// ---- GCode/FB_RestartPrintAction.TcPOU
FUNCTION_BLOCK FB_RestartPrintAction
VAR_INPUT
	bExecute	: BOOL;
END_VAR
VAR_OUTPUT
	bBusy		: BOOL;
	bError		: BOOL;
	nErrorId	: ERRORID;	
END_VAR
VAR_IN_OUT
	stGCodeRef	: ST_GCodeRef;
END_VAR
VAR
	nState		: USINT;
	stAction	: ST_ActionData;
	stError		: ST_Error;
	timer		: TON;
	pTool		: POINTER TO ST_GCodeTool;
END_VAR

IF bExecute THEN
	CASE nState OF
		0:
			bBusy := TRUE;
			MEMSET(ADR(stAction),0,SIZEOF(stAction));
			IF stGCodeRef.pCurrentTool = 0 THEN
				nErrorId := E_ErrorIdGCode.ERRORID_NoSelectedTool;
				bBusy := FALSE;
				bError := FALSE;
			ELSE
				pTool := ADR(stGCodeRef.aToolTable[stGCodeRef.sNciToPlc.Tool]);
				CASE stGCodeRef.pCurrentTool^.P_eObjectType OF
					E_ObjectType.OBJECTTYPE_CartDispenser,
					E_ObjectType.OBJECTTYPE_CartDispStirrer:
						stAction.eAction := E_Action.ACTION_SwitchPressure;
						IF pTool^.bIsInAction1 THEN
							stAction.aParams[1] := 1; //On
							nErrorId := stGCodeRef.pCurrentTool^.M_ExeAction(stAction);
							IF nErrorId > 0 THEN
								nState := 99;
							END_IF
						END_IF
					E_ObjectType.OBJECTTYPE_MultiCartHolder:
						stAction.eAction := E_Action.ACTION_SwitchPressure;
						stAction.aParams[1].0 := pTool^.bIsInAction1;
						stAction.aParams[1].1 := pTool^.bIsInAction2;
						stAction.aParams[1].2 := pTool^.bIsInAction3; 
						nErrorId := stGCodeRef.pCurrentTool^.M_ExeAction(stAction);
						IF nErrorId > 0 THEN
							nState := 99;
						END_IF
					E_ObjectType.OBJECTTYPE_Exposure:
						stAction.eAction := E_Action.ACTION_Expose;
					E_ObjectType.OBJECTTYPE_DeloDot:
						stAction.eAction := E_Action.ACTION_DispenseDrops;
					E_ObjectType.OBJECTTYPE_PiezoPip:
						stAction.eAction := E_Action.ACTION_DispenseDrops;
						stAction.aParams[1] := 0; //Restart macht nur Sinn bei Dauerdispensen
						stAction.aParams[2] := 1;
						nErrorId := stGCodeRef.pCurrentTool^.M_ExeAction(stAction);
						IF nErrorId > 0 THEN
							nState := 99;
						END_IF
					E_ObjectType.OBJECTTYPE_PassivPip,
					E_ObjectType.OBJECTTYPE_Luer:
						nErrorId := stGCodeRef.pCurrentTool^.M_StartUniDispense(0, 0); //beide Parameter auf 0 weil Restart, somit wird der alte Flow verwendet
						IF nErrorId > 0 THEN
							nState := 99;
						END_IF
					E_ObjectType.OBJECTTYPE_Extruder:
						stAction.eAction := E_Action.ACTION_Extrude;
						stAction.aParams[1] := 0;
						stAction.aParams[2] := 1;
						nErrorId := stGCodeRef.pCurrentTool^.M_ExeAction(stAction);
						IF nErrorId > 0 THEN
							nState := 99;
						END_IF
					E_ObjectType.OBJECTTYPE_HybridDispenser:
						stAction.eAction := E_Action.ACTION_BasicDispense;
						stAction.aParams[1] := 1;
						nErrorId := stGCodeRef.pCurrentTool^.M_ExeAction(stAction);
						IF nErrorId > 0 THEN
							nState := 99;
						END_IF
				END_CASE
			END_IF
			IF pTool^.tDelayStart > T#0S THEN
				timer(IN:= TRUE, PT:= pTool^.tDelayStart);
				nState := 1;
			ELSE
				nState := 80;
				bBusy := FALSE;
			END_IF
			
		1:	//Warten auf Timer
			timer();
			IF timer.Q THEN
				bBusy := FALSE;
			END_IF
	END_CASE
	
	IF nState = 99 THEN
		bBusy := FALSE;
		bError := TRUE;
	END_IF
ELSE
	bBusy := FALSE;
	bError := FALSE;
	nErrorId := 0;
	nState := 0;
	timer(IN:=FALSE);
END_IF

END_FUNCTION_BLOCK

// ---- Functions/F_Sub3DPoints.TcPOU
FUNCTION F_Sub3DPoints : ST_3DPoint
VAR_INPUT
	stPoint1	: ST_3DPoint;
	stPoint2	: ST_3DPoint;
END_VAR
VAR
	_stPoint	: ST_3DPoint;
END_VAR

_stPoint.X := stPoint1.X - stPoint2.X;
_stPoint.Y := stPoint1.Y - stPoint2.Y;
_stPoint.Z := stPoint1.Z - stPoint2.Z;
F_Sub3DPoints := _stPoint;

END_FUNCTION

// ---- MainProgs/MAIN.TcPOU
PROGRAM MAIN
VAR
	i				: UINT;
	fbUPS 			: FB_S_UPS;
	fbGetSystemTime : GETSYSTEMTIME;
	bInhibitSequInfo: BOOL;
	nErrInhibitCnt 	: UINT;
	nState			: USINT;
	
	iter : FB_ObjCollectIterator;
	pObject : POINTER TO FB_Object;
	
	(*fbRouterStatusInfo : FB_GetRouterStatusInfo();
	info   : ST_TcRouterStatusInfo;*)

END_VAR

//Sytemzeit ermitteln
fbGetSystemTime(timeLoDW=>timeStamp.dwLowDateTime, timeHiDW=>timeStamp.dwHighDateTime );
//Stromausfall überwachen
fbUPS(iPLCPort:= 851);

(*fbRouterStatusInfo(bExecute:= TRUE);
IF NOT fbRouterStatusInfo.bBusy THEN
	info := fbRouterStatusInfo.info;
	fbRouterStatusInfo(bExecute:= FALSE);
END_IF*)

CASE nState OF
	0:	fbErrorList.A_Reset();
		fbObjectDirectory.M_Init();
		nState := 1;
		//SimutateHwModules();
		//nState := 2;
		
	1:	ScanHwModules();
		IF NOT ScanHwModules.bBusy THEN
			IF ScanHwModules.bError THEN
				//MainDispacher in ErrorState setzen!!
				MainDispacher.M_ForceError();
				nState := 99;
			ELSE
				nState := 2;
			END_IF
		END_IF
		
	2:	//Running
		A_Running();
	
	99:	//In diesem State ist nur FirmwareUpdate möglich
		PC_Control();
		MainDispacher();
		
END_CASE

	
//Nächsten Error aus Errorlist holen (alle 100ms bzw. 10 Zyklen)
//Wenn ein Fehler ausgewertet wurde, dann den nächsten erst wieder nach 10 Zyklen auswerten
//Wenn ein Error zurückgegeben wird, dann wird dieser in stNotifyError geschrieben.
//-> Notification-Variable, welche bei Änderung and GUI gesendet wird.
nErrInhibitCnt := SHR(nErrInhibitCnt,1);
IF fbErrorList.nCount > 0 AND nErrInhibitCnt = 0 THEN
	fbErrorList.A_Get(getValue=> stNotifyError);
	fbErrorList.A_Remove();
	nErrInhibitCnt := 512;
END_IF
//Nächste Info aus SequenceInfoList holen (alle 2 Zyklen)
//Wenn eine SequenceInfo zurückgegeben wurde, dann wird diese in stSequenzInfo geschrieben.
//-> Notification-Variable, welche bei Änderung and GUI gesendet wird.
bInhibitSequInfo := NOT bInhibitSequInfo;
IF bInhibitSequInfo THEN
	fbSequenceInfo.M_GetHead(stSequenceStatus:=stSequenceInfo);		
END_IF

ACTION A_Running:
PC_Control();

MainDispacher();

fbSettings();

ActionDispacher();

fbComplexAction();

IF fbConfiguration.P_bActivated THEN
	//Wird nur aufgerufen, um die Kollisionshöhe bei Bedarf neu zu berechnen
	afbWorkplate[1]();
	
	//Alle Devices aufrufen
	fbObjectDirectory.P_pDeviceCollection^.M_GetIterator(iter);
	WHILE iter.pNode > 0 DO
		pObject := iter.pNode^.P_pObject; 
		pObject^();
		iter.M_Increment();
	END_WHILE
	
	IF afbDryPad[1].P_nObjectID > 0 THEN
		afbDryPad[1].M_UpdateProcessData();
	END_IF
	
END_IF

PerformHardware();
END_ACTION

END_PROGRAM

// ---- Hardware/ScanHwModules.TcPOU
PROGRAM ScanHwModules
VAR
	fbCxGetDeviceIdent	: FB_CxGetDeviceIdentificationEx;
	stDeviceIdentEx		: ST_CxDeviceIdentificationEx;	
	fbGetDeviceIds		: IOF_GetDeviceIDs;
	fbGetDeviceType		: IOF_GetDeviceType;
	fbGetDeviceNetId	: IOF_GetDeviceNetId;
	fbEcGetConfSlaves 	: FB_EcGetConfSlaves;
	fbEcCoeSdoRead		: FB_EcCoESdoRead;

	aDevIds				: ARRAY[0..cMaxDeviceIds - 1] OF WORD;
	nCntEcMaster		: USINT; //Anzahl der gefundenen EtherCAT-Master
	wDevIdCANMaster		: WORD;
	dwBuffer			: DWORD;
	aEtherCATMaster		: ARRAY [1..cMaxEcMaster] OF ST_EtherCATMaster;
	
	nDriveCounter		: USINT;
	aDriveType			: ARRAY[0..3] OF STRING(15);
	aDriveAdsAddr		: ARRAY[0..3] OF ST_AdsAdress;
	
	stCanMasterAddress	: ST_CanMasterAddress;
	bCANInterfaceAvailable	: BOOL;
	nCanNodeCnt			: USINT;
	
	i 					: USINT;
	j					: UINT;
	nState 				: USINT;
	stError				: ST_Error;
	stErrorTmp			: ST_Error;
	bErrorTmp			: BOOL;
	
	nYAxes				: USINT;
	nMultiZRefs			: USINT;

	pYDrive				: POINTER TO FB_XYDriveBase;
	pHwModule			: POINTER TO FB_HwModule;
	pMultiZ				: POINTER TO FB_MultiZRef;
	stHwInfo			: ST_HardwareInfo;
	stHardwareId 		: ST_HardwareId;
	
	test				: UINT;
	
END_VAR
VAR_OUTPUT
	bBusy 	 : BOOL;
	bError	 : BOOL;
	nErrorId : ERRORID;
END_VAR

VAR CONSTANT
	cMaxDeviceIds : USINT := 5;
	cMaxEcMaster : USINT := 2;
END_VAR

stError.POUState := nState;
CASE nState OF
	0:	//PlcInformationen auslesen
		bBusy := TRUE;
		fbCxGetDeviceIdent(bExecute:= TRUE,stDevIdent=>stDeviceIdentEx); //PlcInfo auslesen
		IF NOT fbCxGetDeviceIdent.bBusy THEN
			IF fbCxGetDeviceIdent.bError THEN
				stError.ErrorId := UDINT_TO_UINT(fbCxGetDeviceIdent.nErrorID);
				nState := 99;
			ELSE
				fbCxGetDeviceIdent(bExecute:= FALSE);
				stPlcInfo.sTargetType := stDeviceIdentEx.strTargetType;
				stPlcInfo.sSerialNo := stDeviceIdentEx.strHardwareSerialNo;
				stPlcInfo.sTwinCATBuild := stDeviceIdentEx.strTwinCATBuild;
				stPlcInfo.sPlcVersion := stLibVersion_SPS_PlattformCD.sVersion;
				nState := 1;			
			END_IF
			fbCxGetDeviceIdent(bExecute:= FALSE);
		END_IF

	1:	//Alle DeviceIds abrufen
		fbGetDeviceIds(LEN:= SIZEOF(aDevIds), DESTADDR:= ADR(aDevIds), START:= TRUE); 
		IF NOT fbGetDeviceIds.BUSY THEN
			IF fbGetDeviceIds.ERR THEN
				stError.ErrorId := UDINT_TO_UINT(fbGetDeviceIds.ERRID);
				nState := 99;
			ELSE
				nState := 2;				
			END_IF
			fbGetDeviceIds(START:= FALSE);
		END_IF	

	2:	//DeviceId des EcMasters ermitteln
		fbGetDeviceType(DEVICEID:= aDevIds[i],  START:= TRUE);
		IF NOT fbGetDeviceType.BUSY THEN
			IF fbGetDeviceType.IODeviceType = IODEVICETYPE_ETHERCAT THEN
				nCntEcMaster := nCntEcMaster + 1;
				aEtherCATMaster[nCntEcMaster].nDeviceId := aDevIds[i];;
			ELSIF fbGetDeviceType.IODeviceType = IODEVICETYPE_EL6751 THEN
				wDevIdCANMaster := aDevIds[i];
			END_IF
			i:= i + 1;
			fbGetDeviceType(START:= FALSE);
		END_IF

		IF i > cMaxDeviceIds THEN
			IF aEtherCATMaster[1].nDeviceId = 0 THEN	//es muss mind. 1 EtherCAT-Master gefunden werden
				stError.ErrorId := E_ErrorIdObjMgmt.ERRORID_EtherCATMasterNotConfigured;
				nState := 99;
			ELSIF wDevIdCANMaster = 0 THEN
				stError.ErrorId := E_ErrorIdObjMgmt.ERRORID_CANopenMasterNotConfigured;
				nState := 99;
			ELSE
				nState := 3;
			END_IF
		END_IF
		
	3:	//NetId's der EtherCAT-Master ermitteln
		//wird für jeden Master durchlaufen
		fbGetDeviceNetId(DEVICEID:= aEtherCATMaster[nCntEcMaster].nDeviceId, START:= TRUE, DeviceNetId=> aEtherCATMaster[nCntEcMaster].sNetId);
		IF NOT fbGetDeviceNetId.BUSY THEN
			IF fbGetDeviceNetId.ERR THEN
				stError.ErrorId := UDINT_TO_UINT(fbGetDeviceNetId.ERRID);
				nState := 99;
			ELSE
				nCntEcMaster := nCntEcMaster - 1;
				IF nCntEcMaster = 0 THEN
					nCntEcMaster := nCntEcMaster + 1;
					nState := 4;
				END_IF
			END_IF
			fbGetDeviceNetId(START:= FALSE);
		END_IF
		
	4:	//NetId vom CANopen-Master ermitteln (es ist nur ein Master vorgesehen)
		fbGetDeviceNetId(DEVICEID:= wDevIdCANMaster, START:= TRUE, DeviceNetId=> stCanMasterAddress.sOwnNetId);
		IF NOT fbGetDeviceNetId.BUSY THEN
			IF fbGetDeviceNetId.ERR THEN
				stError.ErrorId := UDINT_TO_UINT(fbGetDeviceNetId.ERRID);
				nState := 99;
			ELSE
				nState := 5;
			END_IF
			fbGetDeviceNetId(START:= FALSE);
		END_IF
		
	5:	//Konfigurierte EtherCAT-Slaves ermitteln und in entsprechendes Array speichern
		//wird für jeden Master durchlaufen
		fbEcGetConfSlaves(sNetId:= aEtherCATMaster[nCntEcMaster].sNetId, pArrEcConfSlaveInfo:= ADR(aEtherCATMaster[nCntEcMaster].aStSlaveInfo),
							cbBufLen:= SIZEOF(aEtherCATMaster[nCntEcMaster].aStSlaveInfo), bExecute:= TRUE, nSlaves=> aEtherCATMaster[nCntEcMaster].nCfgSlaves);
 		IF NOT fbEcGetConfSlaves.bBusy THEN
			IF fbEcGetConfSlaves.bError THEN
				stError.ErrorId := UDINT_TO_UINT(fbEcGetConfSlaves.nErrorId);
				nState := 99;
			ELSE
				IF nCntEcMaster = cMaxEcMaster OR (aEtherCATMaster[nCntEcMaster + 1].sNetId = '') THEN
					nState := 6;
				ELSE
					nCntEcMaster := nCntEcMaster + 1;
				END_IF
			END_IF
			fbEcGetConfSlaves(bExecute := FALSE);
		END_IF
 
	6:	//EtherCAT-Slaves auswerten
		FOR i:= 1 TO nCntEcMaster BY 1 DO
			FOR j:= 0 TO aEtherCATMaster[i].nCfgSlaves BY 1 DO
				IF M_IsXYDrive(aEtherCATMaster[i].aStSlaveInfo[j]) THEN
					aDriveType[nDriveCounter] := aEtherCATMaster[i].aStSlaveInfo[j].sType;
					aDriveAdsAddr[nDriveCounter].sNetId := aEtherCATMaster[i].sNetId;
					aDriveAdsAddr[nDriveCounter].nPort := aEtherCATMaster[i].aStSlaveInfo[j].nAddr;
					nDriveCounter := nDriveCounter + 1;
				ELSIF aEtherCATMaster[i].aStSlaveInfo[j].sType = 'EL6751' THEN
					stCanMasterAddress.sEcMasterNetId := aEtherCATMaster[i].sNetId;
					stCanMasterAddress.nBoxAddress := aEtherCATMaster[i].aStSlaveInfo[j].nAddr;
				ELSIF aEtherCATMaster[i].aStSlaveInfo[j].sType = 'EL6900' OR aEtherCATMaster[i].aStSlaveInfo[j].sType = 'EL1918' THEN
					pFbSafety := ADR(fbSafety);
				ELSIF aEtherCATMaster[i].aStSlaveInfo[j].sType = 'EL7031' OR aEtherCATMaster[i].aStSlaveInfo[j].sType = 'EL7041' OR 
																			aEtherCATMaster[i].aStSlaveInfo[j].sType = 'EL7047' THEN
					{IF defined(variable:fbHwRefSpinDrive)}
						fbHwRefSpinDrive.P_sNetId := aEtherCATMaster[i].sNetId;
					{END_IF}
					{IF defined(variable:fbHwRefLiftDrive)}
						fbHwRefLiftDrive.P_sNetId := aEtherCATMaster[i].sNetId;
					{END_IF}
					{IF defined(variable:fbHwRefTrayStop)}
						fbHwRefTrayStop.P_sNetId := aEtherCATMaster[i].sNetId;
					{END_IF}
				END_IF
			END_FOR
		END_FOR
		
		IF pFbSafety = 0 THEN //kein InterlockSafe
			//SimpleInterlock möglich?
			IF F_GetMappingStatus(ADR(fbSafetyPseudo.bInput),SIZEOF(fbSafetyPseudo.bInput)) = EPlcMappingStatus.MS_Partial THEN
				pFbSafety := ADR(fbSafetyPseudo);
			ELSE
				pFbSafety := ADR(fbSafetyBase); //Dummy
			END_IF
		ELSE
			fbSafety.M_CheckBoxCtcMapping();
		END_IF
		
		//XYDrive-Pointer den entsprechenden XYDrive-Instanzen zuordnen
		IF aDriveType[0] = 'EL7041' AND aDriveType[1] = 'EL7041' AND aDriveType[2] = 'EL7041' THEN	//Plattform C
			//X
			stHardwareId.eGroup := E_HardwareGrp.AxisX;
			stHardwareId.nParentItem := 0;
			stHardwareId.nItem := 1;
			fbXDriveBeck.P_stHardwareId := stHardwareId;
			fbXDriveBeck.P_stAdsAddress := aDriveAdsAddr[0];
			fbXYDriveList.M_Add(ADR(fbXDriveBeck));
			//Y
			stHardwareId.eGroup := E_HardwareGrp.AxisY;
			stHardwareId.nParentItem := 1;
			stHardwareId.nItem := 1;
			fbYDriveBeck.P_stHardwareId := stHardwareId;
			fbYDriveBeck.P_stAdsAddress := aDriveAdsAddr[2];
			fbXYDriveList.M_Add(ADR(fbYDriveBeck));
			nYAxes := 1;
			
			stTipCalibrator.bInvert := FALSE;
			
		ELSIF  (LEFT(aDriveType[0],11) = 'C1150-DS-XC' AND LEFT(aDriveType[1],11) = 'C1150-DS-XC' AND LEFT(aDriveType[2],11) = 'C1150-DS-XC') THEN //Plattform D zwei Ebenen

			stHardwareId.eGroup := E_HardwareGrp.AxisX;
			stHardwareId.nParentItem := 0;
			stHardwareId.nItem := 1;
			fbX1DriveLmtDS.P_stHardwareId := stHardwareId;
			fbX1DriveLmtDS.P_stAdsAddress := aDriveAdsAddr[2];
			fbXYDriveList.M_Add(ADR(fbX1DriveLmtDS));
			
			stHardwareId.eGroup := E_HardwareGrp.AxisY;
			stHardwareId.nParentItem := 1;
			stHardwareId.nItem := 1;
			fbY1DriveLmtDS.P_stHardwareId := stHardwareId;
			fbY1DriveLmtDS.P_stAdsAddress := aDriveAdsAddr[0];
			fbXYDriveList.M_Add(ADR(fbY1DriveLmtDS));
			
			stHardwareId.eGroup := E_HardwareGrp.AxisY;
			stHardwareId.nParentItem := 1;
			stHardwareId.nItem := 2;
			fbY2DriveLmtDS.P_stHardwareId := stHardwareId;
			fbY2DriveLmtDS.P_stAdsAddress := aDriveAdsAddr[1];
			fbXYDriveList.M_Add(ADR(fbY2DriveLmtDS));
			nYAxes := 2;
			
			stTipCalibrator.bInvert := FALSE;
			
		ELSIF (LEFT(aDriveType[0],11) = 'C1250-DS-XC' AND LEFT(aDriveType[1],11) = 'C1250-DS-XC' AND LEFT(aDriveType[2],11) = 'C1250-DS-XC') THEN  //Plattform D zwei Ebenen
			stHardwareId.eGroup := E_HardwareGrp.AxisX;
			stHardwareId.nParentItem := 0;
			stHardwareId.nItem := 1;
			fbX1DriveLmtDS.P_stHardwareId := stHardwareId;
			fbX1DriveLmtDS.P_stAdsAddress := aDriveAdsAddr[0];
			fbXYDriveList.M_Add(ADR(fbX1DriveLmtDS));
			
			stHardwareId.eGroup := E_HardwareGrp.AxisY;
			stHardwareId.nParentItem := 1;
			stHardwareId.nItem := 1;
			fbY1DriveLmtDS.P_stHardwareId := stHardwareId;
			fbY1DriveLmtDS.P_stAdsAddress := aDriveAdsAddr[2];
			fbXYDriveList.M_Add(ADR(fbY1DriveLmtDS));
			
			stHardwareId.eGroup := E_HardwareGrp.AxisY;
			stHardwareId.nParentItem := 1;
			stHardwareId.nItem := 2;
			fbY2DriveLmtDS.P_stHardwareId := stHardwareId;
			fbY2DriveLmtDS.P_stAdsAddress := aDriveAdsAddr[1];
			fbXYDriveList.M_Add(ADR(fbY2DriveLmtDS));

			stTipCalibrator.bInvert := TRUE;
			
			nYAxes := 2;
			
		ELSIF (LEFT(aDriveType[0],11) = 'C1100-EC-XC' AND LEFT(aDriveType[1],11) = 'C1100-EC-XC' AND LEFT(aDriveType[2],11) = 'C1100-EC-XC') THEN
			stHardwareId.eGroup := E_HardwareGrp.AxisX;
			stHardwareId.nParentItem := 0;
			stHardwareId.nItem := 1;
			fbX1DriveLmtEC.P_stHardwareId := stHardwareId;
			fbX1DriveLmtEC.P_stAdsAddress := aDriveAdsAddr[0];
			fbXYDriveList.M_Add(ADR(fbX1DriveLmtEC));
			
			stHardwareId.eGroup := E_HardwareGrp.AxisY;
			stHardwareId.nParentItem := 1;
			stHardwareId.nItem := 1;
			fbY1DriveLmtEC.P_stHardwareId := stHardwareId;
			fbY1DriveLmtEC.P_stAdsAddress := aDriveAdsAddr[1];
			fbXYDriveList.M_Add(ADR(fbY1DriveLmtEC));
			
			stHardwareId.eGroup := E_HardwareGrp.AxisY;
			stHardwareId.nParentItem := 1;
			stHardwareId.nItem := 2;
			fbY2DriveLmtEC.P_stHardwareId := stHardwareId;
			fbY2DriveLmtEC.P_stAdsAddress := aDriveAdsAddr[2];
			fbXYDriveList.M_Add(ADR(fbY2DriveLmtEC));
			nYAxes := 2;
			
		ELSIF (LEFT(aDriveType[0],11) = 'C1150-DS-XC' AND LEFT(aDriveType[1],11) = 'C1150-DS-XC') OR
				(LEFT(aDriveType[0],11) = 'C1250-DS-XC' AND LEFT(aDriveType[1],11) = 'C1250-DS-XC') THEN //Plattform D eine Ebene
			stHardwareId.eGroup := E_HardwareGrp.AxisX;
			stHardwareId.nParentItem := 0;
			stHardwareId.nItem := 1;
			fbX1DriveLmtDS.P_stHardwareId := stHardwareId;
			fbX1DriveLmtDS.P_stAdsAddress := aDriveAdsAddr[0];
			fbXYDriveList.M_Add(ADR(fbX1DriveLmtDS));
			
			stHardwareId.eGroup := E_HardwareGrp.AxisY;
			stHardwareId.nParentItem := 1;
			stHardwareId.nItem := 1;
			fbY1DriveLmtDS.P_stHardwareId := stHardwareId;
			fbY1DriveLmtDS.P_stAdsAddress := aDriveAdsAddr[1];
			fbXYDriveList.M_Add(ADR(fbY1DriveLmtDS));
			nYAxes := 1;
			
			//Bei der C1150 wird das Signal nicht invertiert
			IF LEFT(aDriveType[0],11) = 'C1250-DS-XC' THEN
				stTipCalibrator.bInvert := TRUE;
			ELSE
				stTipCalibrator.bInvert := FALSE;
			END_IF

		ELSE
			stError.ErrorId := E_ErrorIdObjMgmt.ERRORID_InvalidDriveConfig;
			nState := 99;
			RETURN;
		END_IF
		
		nState := 8;
		
	8:	//Überprüfen, welche CAN-Nodes im CANopen-Master konfiguriert - Schritt 1
		//Konfiguration steht in COE-Objektverzeichnis 8000h-87E0h Subindex 0 des CANopen-Masters
		fbEcCoeSdoRead(sNetId:= stCanMasterAddress.sEcMasterNetId, nSlaveAddr:= stCanMasterAddress.nBoxAddress, nIndex:= 16#8000 + 16 * nCanNodeCnt, nSubIndex:= 0,
					pDstBuf:= ADR(dwBuffer), cbBufLen:= 2, bExecute:= TRUE);
					
		IF NOT fbEcCoeSdoRead.bBusy THEN
			IF fbEcCoeSdoRead.bError THEN
				stError.ErrorId := UDINT_TO_UINT(fbEcCoeSdoRead.nErrId);
				nState := 99;
			ELSE
				//Wenn 36 ist Node ein CAN-Interface, wenn 46, dann ein CANopen-Slave
				//Das CAN-Interface steht immer an erster Stelle, es wird aber nach dem letzten CANopen-Node abermals eine 36 zurückgegeben
				IF dwBuffer = 36 AND NOT bCANInterfaceAvailable THEN //CAN-Interface
					nCanNodeCnt := nCanNodeCnt + 1;
					bCANInterfaceAvailable := TRUE;
				ELSIF dwBuffer = 46 THEN //CANopen-Node
					nState := 9;
				ELSE
					nState := 10;
				END_IF
			END_IF
			fbEcCoeSdoRead(bExecute:= FALSE);
		END_IF
		
	9:	//Überprüfen, welche CANopen-Nodes im CANopen-Master konfiguriert - Schritt 2
		//NodeAdress steht in COE-Objektverzeichnis 8000h-87E0h Subindex 1 des CANopen-Masters
		fbEcCoeSdoRead(sNetId:= stCanMasterAddress.sEcMasterNetId, nSlaveAddr:= stCanMasterAddress.nBoxAddress, nIndex:= 16#8000 + 16 * nCanNodeCnt, nSubIndex:= 1,
					pDstBuf:= ADR(dwBuffer), cbBufLen:= 2, bExecute:= TRUE);
					
		IF NOT fbEcCoeSdoRead.bBusy THEN
			IF fbEcCoeSdoRead.bError THEN
				stError.ErrorId := UDINT_TO_UINT(fbEcCoeSdoRead.nErrId);
				nState := 99;
			ELSE
				IF dwBuffer = 0 OR nCanNodeCnt = 126 THEN
					nState := 10; //kein weiterer Node vorhanden
				ELSE
					aCanNodes[dwBuffer] := TRUE;
					nState := 8; //zurück zu Schritt 1 (nState 8)
					nCanNodeCnt := nCanNodeCnt + 1;
				END_IF
			END_IF
			fbEcCoeSdoRead(bExecute:= FALSE);
		END_IF
		
	10:	//Zuordung der CAN-Node-Ids zu den HwModul-Referenzen
		//Tip-Cleaner nimmt eine Sonderstellung ein, da er kein Gesim-CANopen-Node ist
		stTipCleanerRef.stAdsAdress.sNetId := stCanMasterAddress.sOwnNetId;
		stTipCleanerRef.stAdsAdress.nPort := 36 + 4096; //36=NodeId
		
		//MultiZ
		FOR i := 1 TO cMaxMzHeads BY 1 DO
			IF aCanNodes[i + 7] THEN
				afbMultiZRef[i].M_Prepare(stCanMasterAddress.sOwnNetId ,nCanNodeId := UINT_TO_USINT(i + 7));
				fbMultiZRefList.M_Add(ADR(afbMultiZRef[i]));
				fbCANOpenHwModuleList.M_Add(ADR(afbMultiZRef[i]));
				nMultiZRefs := nMultiZRefs + 1;
			END_IF
		END_FOR
		
		//Zuordung der MultiZRefs zu den XY-Drives
		fbMultiZRefList.M_SetCurrentToHead();
		IF nYAxes = 1 THEN
			stHardwareId.eGroup := E_HardwareGrp.AxisY;
			stHardwareId.nParentItem := 1;	//derzeit gibt es nur eine X-Achse
			stHardwareId.nItem := 1;
			pYDrive := fbXYDriveList.M_GetByHwId(stHardwareId);
			IF pYDrive > 0 THEN
				pYDrive^.P_pMultiZRef := fbMultiZRefList.M_Get();
				stHardwareId.eGroup := E_HardwareGrp.MultiZBasis;
				stHardwareId.nParentItem := 1;
				stHardwareId.nItem := 1;
				pYDrive^.P_pMultiZRef^.P_stHardwareId := stHardwareId;
			END_IF
		ELSIF nYAxes = 2 AND nMultiZRefs = 1 THEN
			stHardwareId.eGroup := E_HardwareGrp.AxisY;
			stHardwareId.nParentItem := 1;	//derzeit gibt es nur eine X-Achse
			stHardwareId.nItem := 2;
			pYDrive := fbXYDriveList.M_GetByHwId(stHardwareId);
			IF pYDrive > 0 THEN
				pYDrive^.P_pMultiZRef := fbMultiZRefList.M_Get();
				stHardwareId.eGroup := E_HardwareGrp.MultiZBasis;
				stHardwareId.nParentItem := 2;
				stHardwareId.nItem := 1;
				pYDrive^.P_pMultiZRef^.P_stHardwareId := stHardwareId;
			END_IF
		ELSIF nYAxes = 2 AND nMultiZRefs = 2 THEN
			stHardwareId.eGroup := E_HardwareGrp.AxisY;
			stHardwareId.nParentItem := 1;	//derzeit gibt es nur eine X-Achse
			stHardwareId.nItem := 1;
			pYDrive := fbXYDriveList.M_GetByHwId(stHardwareId);
			IF pYDrive > 0 THEN
				pYDrive^.P_pMultiZRef := fbMultiZRefList.M_Get(); 
				stHardwareId.eGroup := E_HardwareGrp.MultiZBasis;
				stHardwareId.nParentItem := 1;
				stHardwareId.nItem := 1;
				pYDrive^.P_pMultiZRef^.P_stHardwareId := stHardwareId;
			END_IF
			stHardwareId.eGroup := E_HardwareGrp.AxisY;
			stHardwareId.nParentItem := 1;	//derzeit gibt es nur eine X-Achse
			stHardwareId.nItem := 2;
			pYDrive := fbXYDriveList.M_GetByHwId(stHardwareId);
			IF pYDrive > 0 THEN
				pYDrive^.P_pMultiZRef := fbMultiZRefList.M_Get();
				stHardwareId.eGroup := E_HardwareGrp.MultiZBasis;
				stHardwareId.nParentItem := 2;
				stHardwareId.nItem := 2;
				pYDrive^.P_pMultiZRef^.P_stHardwareId := stHardwareId;
 			END_IF			
		END_IF
		
		{IF defined(variable:afbMtpHeatRef)}
		FOR i := 0 TO (cNoOfMtpHeaters  - 1) BY 1 DO
			IF aCanNodes[i + cNodeIdMtpHeater1] THEN
				stHardwareId.eGroup := E_HardwareGrp.MtpHeater;
				stHardwareId.nParentItem := 0;
				stHardwareId.nItem := i + 1;
				afbMtpHeatRef[i + 1].P_stHardwareId := stHardwareId;
				afbMtpHeatRef[i + 1].M_Prepare(stCanMasterAddress.sOwnNetId ,nCanNodeId := UINT_TO_USINT(i + cNodeIdMtpHeater1));
				afbMtpHeatRef[i + 1]();
				fbCANOpenHwModuleList.M_Add(ADR(afbMtpHeatRef[i + 1]));
			END_IF
		END_FOR
		{END_IF}
		
		{IF defined(variable:afbSubstHeatRef)}
		FOR i := 0 TO (cNoOfSubstHeaters - 1) BY 1 DO
			IF aCanNodes[i + cNodeIdSubstHeater1] THEN
				stHardwareId.eGroup := E_HardwareGrp.SubstHeater;
				stHardwareId.nParentItem := 0;
				stHardwareId.nItem := i + 1;
				afbSubstHeatRef[i + 1].P_stHardwareId := stHardwareId;
				afbSubstHeatRef[i + 1].M_Prepare(stCanMasterAddress.sOwnNetId ,nCanNodeId := UINT_TO_USINT(i + cNodeIdSubstHeater1));
				afbSubstHeatRef[i + 1]();
				fbCANOpenHwModuleList.M_Add(ADR(afbSubstHeatRef[i + 1]));
			END_IF
		END_FOR
		{END_IF}
		
		{IF defined(variable: aFbReactDriveRef)}
		FOR i := 0 TO (cNoOfReactDrives - 1) BY 1 DO
			IF aCanNodes[i + cNodeIdReactDrive1] THEN
				stHardwareId.eGroup := E_HardwareGrp.ReactorDrive;
				stHardwareId.nParentItem := 0;
				stHardwareId.nItem := i + 1;
				aFbReactDriveRef[i + 1].P_stHardwareId := stHardwareId;			
				aFbReactDriveRef[i + 1].M_Prepare(stCanMasterAddress.sOwnNetId ,nCanNodeId := UINT_TO_USINT(i + cNodeIdReactDrive1));
				aFbReactDriveRef[i + 1]();
				fbCANOpenHwModuleList.M_Add(ADR(aFbReactDriveRef[i + 1]));
			END_IF
		END_FOR
		{END_IF}

		{IF defined(variable: aFbReactHeatRef)}
		FOR i := 0 TO (cNoOfReactHeaters - 1) BY 1 DO
			IF aCanNodes[i + cNodeIdReactHeater1] THEN
				stHardwareId.eGroup := E_HardwareGrp.ReactorHeater;
				stHardwareId.nParentItem := 0;
				stHardwareId.nItem := i + 1;
				aFbReactHeatRef[i + 1].P_stHardwareId := stHardwareId;			
				aFbReactHeatRef[i + 1].M_Prepare(stCanMasterAddress.sOwnNetId ,nCanNodeId := UINT_TO_USINT(i + cNodeIdReactHeater1));
				aFbReactHeatRef[i + 1]();
				fbCANOpenHwModuleList.M_Add(ADR(aFbReactHeatRef[i + 1]));
			END_IF
		END_FOR
		{END_IF}
		
		{IF defined(variable:aFbTripleTriggerRef)}
		FOR i := 0 TO (cNoOfTripleTriggers - 1) BY 1 DO
			IF aCanNodes[i + cNodeIdTripleTrigger1] THEN
				stHardwareId.eGroup := E_HardwareGrp.TripleTrigger;
				stHardwareId.nParentItem := 0;
				stHardwareId.nItem := i + 1;
				aFbTripleTriggerRef[i + 1].P_stHardwareId := stHardwareId;			
				aFbTripleTriggerRef[i + 1].M_Prepare(stCanMasterAddress.sOwnNetId ,nCanNodeId := UINT_TO_USINT(i + cNodeIdTripleTrigger1));
				aFbTripleTriggerRef[i + 1]();
				fbCANOpenHwModuleList.M_Add(ADR(aFbTripleTriggerRef[i + 1]));
			END_IF		
		END_FOR
		{END_IF}
		
		{IF defined(variable:aFbIOExpanderRef)}
		FOR i := 0 TO (cNoOfIOExpanders - 1) BY 1 DO
			IF aCanNodes[i + cNodeIdIOExpander1] THEN
				stHardwareId.eGroup := E_HardwareGrp.IOExpander;
				stHardwareId.nParentItem := 0;
				stHardwareId.nItem := i + 1;
				aFbIOExpanderRef[i + 1].P_stHardwareId := stHardwareId;		
				aFbIOExpanderRef[i + 1].M_Prepare(stCanMasterAddress.sOwnNetId ,nCanNodeId := UINT_TO_USINT(i + cNodeIdIOExpander1));
				aFbIOExpanderRef[i + 1]();
				fbCANOpenHwModuleList.M_Add(ADR(aFbIOExpanderRef[i + 1]));
			END_IF
		END_FOR
		{END_IF}
		
		{IF defined(variable:aFbBottleRackRef)}
		FOR i := 0 TO (cNoOfBottleRacks - 1) BY 1 DO
			IF aCanNodes[i + cNodeIdBottleRack1] THEN
				stHardwareId.eGroup := E_HardwareGrp.BottleRack;
				stHardwareId.nParentItem := 0;
				stHardwareId.nItem := i + 1;
				aFbBottleRackRef[i + 1].P_stHardwareId := stHardwareId;			
				aFbBottleRackRef[i + 1].M_Prepare(stCanMasterAddress.sOwnNetId ,nCanNodeId := UINT_TO_USINT(i + cNodeIdBottleRack1));
				aFbBottleRackRef[i + 1]();
				fbCANOpenHwModuleList.M_Add(ADR(aFbBottleRackRef[i + 1]));
			END_IF
		END_FOR
		{END_IF}
		
		
		{IF defined(variable:aFbInkStatDrvSpinRef)}
		FOR i := 0 TO (cNoOfInkStatSpinDrives - 1) BY 1 DO
			IF aCanNodes[i + cNodeIdInkStatSpinDrive1] THEN
				stHardwareId.eGroup := E_HardwareGrp.InkStationSpinDrive;
				stHardwareId.nParentItem := 0;
				stHardwareId.nItem := i + 1;
				aFbInkStatDrvSpinRef[i + 1].P_stHardwareId := stHardwareId;		
				aFbInkStatDrvSpinRef[i + 1].M_Prepare(stCanMasterAddress.sOwnNetId ,nCanNodeId := UINT_TO_USINT(i + cNodeIdInkStatSpinDrive1));
				aFbInkStatDrvSpinRef[i + 1]();
				fbCANOpenHwModuleList.M_Add(ADR(aFbInkStatDrvSpinRef[i + 1]));
			END_IF
		END_FOR
		{END_IF}

		{IF defined(variable:aFbInkStatDrvCoverRef)}
		FOR i := 0 TO (cNoOfInkStatCoverDrives - 1) BY 1 DO
			IF aCanNodes[i + cNodeIdInkStatCoverDrive1] THEN
				stHardwareId.eGroup := E_HardwareGrp.InkStationCoverDrive;
				stHardwareId.nParentItem := 0;
				stHardwareId.nItem := i + 1;
				aFbInkStatDrvCoverRef[i + 1].P_stHardwareId := stHardwareId;
				aFbInkStatDrvCoverRef[i + 1].M_Prepare(stCanMasterAddress.sOwnNetId ,nCanNodeId := UINT_TO_USINT(i + cNodeIdInkStatCoverDrive1));
				aFbInkStatDrvCoverRef[i + 1]();
				fbCANOpenHwModuleList.M_Add(ADR(aFbInkStatDrvCoverRef[i + 1]));
			END_IF
		END_FOR
		{END_IF}
		
		{IF defined(variable:aFbPowderStatRef)}
		FOR i := 0 TO (cNoOfPowderStations - 1) BY 1 DO
			IF aCanNodes[i + cNodeIdPowderStation1] THEN
				stHardwareId.eGroup := E_HardwareGrp.PowderStation;
				stHardwareId.nParentItem := 0;
				stHardwareId.nItem := i + 1;
				aFbPowderStatRef[i + 1].P_stHardwareId := stHardwareId;				
				aFbPowderStatRef[i + 1].M_Prepare(stCanMasterAddress.sOwnNetId ,nCanNodeId := UINT_TO_USINT(i + cNodeIdPowderStation1));
				aFbPowderStatRef[i + 1]();
				fbCANOpenHwModuleList.M_Add(ADR(aFbPowderStatRef[i + 1]));
			END_IF
		END_FOR
		{END_IF}
		
		//MulitPurposeIO (F-Einschub)
		{IF defined(variable:aFbHwRefMultiPurpIO)}
		FOR i:= 0 TO (cNoOfMultiPurpIO - 1) BY 1 DO
			IF aCanNodes[i + cNodeIdMultiPurpIO] THEN
				stHardwareId.eGroup := E_HardwareGrp.MultiPurpIO;
				stHardwareId.nParentItem := 0;
				stHardwareId.nItem := i + 1;
				aFbHwRefMultiPurpIO[i + 1].P_stHardwareId := stHardwareId;
				aFbHwRefMultiPurpIO[i + 1].M_Prepare(stCanMasterAddress.sOwnNetId ,nCanNodeId := UINT_TO_USINT(i + cNodeIdMultiPurpIO));
				fbCANOpenHwModuleList.M_Add(ADR(aFbHwRefMultiPurpIO[i + 1]));
			END_IF
		END_FOR
		{END_IF}
		
		//TrayTransporter in 3 verschiedenen Varianten
		{IF defined(TrayTransporterL)}
		stHardwareId.eGroup := E_HardwareGrp.NanotecPD;
		stHardwareId.nParentItem := 0;
		stHardwareId.nItem := 1;
		fbHwRefTrayTransSlider.P_stHardwareId := stHardwareId;
		fbHwRefTrayTransSlider.M_Prepare(stCanMasterAddress.sOwnNetId ,nCanNodeId := 1);
		fbCANOpenHwModuleList.M_Add(ADR(fbHwRefTrayTransSlider));
		stHardwareId.eGroup := E_HardwareGrp.TMCM1140Stepper_Gen2;
		fbHwRefDrivingPinLeft.P_stHardwareId := stHardwareId;
		fbHwRefDrivingPinLeft.M_Prepare(stCanMasterAddress.sOwnNetId ,nCanNodeId := 36);
		fbCANOpenHwModuleList.M_Add(ADR(fbHwRefDrivingPinLeft));
		
		{ELSIF defined(TrayTransporterR)}
		stHardwareId.eGroup := E_HardwareGrp.NanotecPD;
		stHardwareId.nParentItem := 0;
		stHardwareId.nItem := 1;
		fbHwRefTrayTransSlider.P_stHardwareId := stHardwareId;
		fbHwRefTrayTransSlider.M_Prepare(stCanMasterAddress.sOwnNetId ,nCanNodeId := 1);
		fbCANOpenHwModuleList.M_Add(ADR(fbHwRefTrayTransSlider));
		stHardwareId.eGroup := E_HardwareGrp.TMCM1140Stepper_Gen2;
		fbHwRefDrivingPinRight.P_stHardwareId := stHardwareId;
		fbHwRefDrivingPinRight.M_Prepare(stCanMasterAddress.sOwnNetId ,nCanNodeId := 35);
		fbCANOpenHwModuleList.M_Add(ADR(fbHwRefDrivingPinRight));
		
		{ELSIF defined(TrayTransporterLR)}
		stHardwareId.eGroup := E_HardwareGrp.NanotecPD;
		stHardwareId.nParentItem := 0;
		stHardwareId.nItem := 1;
		fbHwRefTrayTransSlider.P_stHardwareId := stHardwareId;
		fbHwRefTrayTransSlider.M_Prepare(stCanMasterAddress.sOwnNetId ,nCanNodeId := 1);
		fbCANOpenHwModuleList.M_Add(ADR(fbHwRefTrayTransSlider));
		stHardwareId.eGroup := E_HardwareGrp.TMCM1140Stepper_Gen2;
		fbHwRefDrivingPinLeft.P_stHardwareId := stHardwareId;
		fbHwRefDrivingPinLeft.M_Prepare(stCanMasterAddress.sOwnNetId ,nCanNodeId := 36);
		fbCANOpenHwModuleList.M_Add(ADR(fbHwRefDrivingPinLeft));
		stHardwareId.nItem := 2;
		fbHwRefDrivingPinRight.P_stHardwareId := stHardwareId;
		fbHwRefDrivingPinRight.M_Prepare(stCanMasterAddress.sOwnNetId ,nCanNodeId := 35);
		fbCANOpenHwModuleList.M_Add(ADR(fbHwRefDrivingPinRight));
		{END_IF}
		
		{IF defined(FDM2)}
		stHardwareId.eGroup := E_HardwareGrp.TMCM1140Stepper_Gen2;
		stHardwareId.nItem := 3;
		fbHwRefFDM_TMCM.P_stHardwareId := stHardwareId;
		//Vielleicht sollte die NodeID mit über M_Init gesetzt werden?
		fbHwRefFDM_TMCM.M_Prepare(stCanMasterAddress.sOwnNetId ,nCanNodeId := 3);
		fbCANOpenHwModuleList.M_Add(ADR(fbHwRefFDM_TMCM));
		{END_IF}
		
		{IF defined(Pure1)}
		stHardwareId.eGroup := E_HardwareGrp.TMCM1140Stepper_Gen2;
		stHardwareId.nItem := 4;
		fbHwRefTMCM_Pure1.P_stHardwareId := stHardwareId;
		//Vielleicht sollte die NodeID mit über M_Init gesetzt werden?
		fbHwRefTMCM_Pure1.M_Prepare(stCanMasterAddress.sOwnNetId ,nCanNodeId := 41);
		fbCANOpenHwModuleList.M_Add(ADR(fbHwRefTMCM_Pure1));
		{END_IF}
		
		{IF defined(Pure2)}
		stHardwareId.eGroup := E_HardwareGrp.TMCM1140Stepper_Gen2;
		stHardwareId.nItem := 5;
		fbHwRefTMCM_Pure2.P_stHardwareId := stHardwareId;
		//Vielleicht sollte die NodeID mit über M_Init gesetzt werden?
		fbHwRefTMCM_Pure2.M_Prepare(stCanMasterAddress.sOwnNetId ,nCanNodeId := 42);
		fbCANOpenHwModuleList.M_Add(ADR(fbHwRefTMCM_Pure2));
		{END_IF}
		
		{IF defined(Pure3)}
		stHardwareId.eGroup := E_HardwareGrp.TMCM1140Stepper_Gen2;
		stHardwareId.nItem := 6;
		fbHwRefTMCM_Pure3.P_stHardwareId := stHardwareId;
		//Vielleicht sollte die NodeID mit über M_Init gesetzt werden?
		fbHwRefTMCM_Pure3.M_Prepare(stCanMasterAddress.sOwnNetId ,nCanNodeId := 43);
		fbCANOpenHwModuleList.M_Add(ADR(fbHwRefTMCM_Pure3));
		{END_IF}
		
		{IF defined(variable:fbHwRefSpinDrive)}
		stHardwareId.eGroup := E_HardwareGrp.EL70xx;
		stHardwareId.nParentItem := 0;
		stHardwareId.nItem := 1;
		fbHwRefSpinDrive.M_Prepare();
		{END_IF}
		{IF defined(variable:fbHwRefLiftDrive)}
		stHardwareId.eGroup := E_HardwareGrp.EL70xx;
		stHardwareId.nParentItem := 0;
		stHardwareId.nItem := 2;
		fbHwRefLiftDrive.M_Prepare();
		{END_IF}
		{IF defined(variable:fbHwRefTrayStop)}
		stHardwareId.eGroup := E_HardwareGrp.EL70xx;
		stHardwareId.nParentItem := 0;
		stHardwareId.nItem := 3;
		fbHwRefTrayStop.M_Prepare();
		{END_IF}
		
		nState := 11;
		
	11:	//Warten, bis alle HwModules ready
		nState := 12;
		fbXYDriveList.M_SetCurrentToHead();
		REPEAT
			pHwModule := fbXYDriveList.M_Get();
			IF pHwModule > 0 THEN
				pHwModule^();
				IF pHwModule^.P_bBusy THEN
					nState := 11;
				END_IF
			END_IF		
		UNTIL pHwModule = 0
		END_REPEAT
		
		fbCANOpenHwModuleList.M_SetCurrentToHead();
		REPEAT
			pHwModule := fbCANOpenHwModuleList.M_Get();
			IF pHwModule > 0 THEN
				pHwModule^();
				IF pHwModule^.P_bBusy THEN
					nState := 11;
				ELSE
					IF pHwModule^.P_bError THEN
						stErrorTmp := pHwModule^.P_stError;
						stError.ErrorId := stErrorTmp.ErrorId;
						stError.ErrorId2 := stErrorTmp.ErrorId2;
						stError.HardwareGrp := stErrorTmp.HardwareGrp;
						stError.HardwareNr := stErrorTmp.HardwareNr;
						bErrorTmp := TRUE;
						EXIT;
					END_IF
				END_IF
			END_IF
		UNTIL pHwModule = 0
		END_REPEAT
		
		{IF defined(variable:fbHwRefSpinDrive)}
		IF fbHwRefSpinDrive.P_bBusy THEN
			nState := 11;
		END_IF
		{END_IF}
		
		{IF defined(variable:fbHwRefLiftDrive)}
		IF fbHwRefLiftDrive.P_bBusy THEN
			nState := 11;
		END_IF
		{END_IF}
		
		{IF defined(variable:fbHwRefTrayStop)}
		IF fbHwRefTrayStop.P_bBusy THEN
			nState := 11;
		END_IF
		{END_IF}
		
		IF bErrorTmp THEN
			nState := 99;
		END_IF
	
	12:	//HwInfoList füllen
		fbCANOpenHwModuleList.M_SetCurrentToHead();
		REPEAT
			pHwModule := fbCANOpenHwModuleList.M_Get();
			IF pHwModule > 0 THEN
				stHwInfo := pHwModule^.M_GetHwInfo();
				HwInfoList.M_Add(stHwInfo);
				IF pHwModule^.P_eHardwareGrp = E_HardwareGrp.MultiZBasis THEN
					pMultiZ := pHwModule;
					FOR i := 1 TO 7 BY 1 DO
						IF pMultiZ^.aFbZAxisRef[i].stInput.nStatus.7 THEN
							pMultiZ^.aFbZAxisRef[i].M_RenewHwId();
							stHwInfo := pMultiZ^.aFbZAxisRef[i].M_GetHwInfo();
							HwInfoList.M_Add(stHwInfo);
						END_IF
					END_FOR
				END_IF
			END_IF
		UNTIL pHwModule = 0
		END_REPEAT
		
		IF bErrorTmp THEN
			nState := 99;
		ELSE
			nState := 80;	
		END_IF
		bBusy := FALSE;
END_CASE

IF nState = 99 THEN
	stError.POU := E_POU.POU_ScanHwModules;
	stError.Cmd := 0;
	stError.POUAction := E_POUACT.POUACT_UNDEFIEND;
	fbErrorList.M_Add(stError);
	bError := TRUE;
	bBusy := FALSE;
END_IF

METHOD M_IsXYDrive : BOOL
VAR_INPUT
	//sDeviceType : STRING(15);
	stSlaveInfo : ST_EcSlaveConfigData;
END_VAR

VAR
	sTemp : STRING(6);
END_VAR
IF FIND(stSlaveInfo.sName, 'P2') > 0 THEN //Die XY-Drive Klemmen sind niemals auf +P2
	RETURN;
END_IF

sTemp := LEFT(stSlaveInfo.sType, 6);
IF sTemp = 'EL7041' OR
	sTemp = 'C1100-' OR
	sTemp = 'C1150-' OR
	sTemp = 'C1250-' THEN
	M_IsXYDrive := TRUE;
END_IF
END_METHOD

END_PROGRAM

// ---- Hardware/HwInfoList.TcPOU
PROGRAM HwInfoList
VAR
	pHead	: POINTER TO ST_Pointer;
	pTail	: POINTER TO ST_Pointer;
	pCurrent: POINTER TO ST_Pointer;	
END_VAR

METHOD FB_exit : BOOL
VAR_INPUT
	bInCopyCode : BOOL; // if TRUE, the exit method is called for exiting an instance that is copied afterwards (online change).
END_VAR

VAR
	pPointer : POINTER TO ST_Pointer;
END_VAR
WHILE pPointer > 0 DO
	__DELETE(pPointer^.pContent);
	__DELETE(pPointer);
	pPointer := pPointer^.pNext;
END_WHILE
END_METHOD

METHOD M_Add
VAR_INPUT
	stHwInfo : ST_HardwareInfo;
END_VAR

VAR
	pNewPointer : POINTER TO ST_Pointer;
	pNewHwInfo : POINTER TO ST_HardwareInfo;
	pModule: POINTER TO PVOID;
END_VAR
pNewPointer := __NEW(ST_Pointer);
MEMSET(pNewPointer,0,SIZEOF(ST_Pointer));
pNewHwInfo := __NEW(ST_HardwareInfo);
pNewHwInfo^ := stHwInfo;

pNewPointer^.pContent := pNewHwInfo;

IF pHead = 0 THEN
	pHead := pTail := pNewPointer;
ELSE
	pNewPointer^.pPrev := pTail; 
	pTail^.pNext := pNewPointer;
	pTail := pNewPointer;
END_IF
END_METHOD

METHOD M_GetNext : ST_HardwareInfo
VAR_INPUT
END_VAR

VAR
	pHwInfo : POINTER TO ST_HardwareInfo;
END_VAR
IF pCurrent > 0 THEN
	pHwInfo := pCurrent^.pContent;
	M_GetNext := pHwInfo^;
	pCurrent := pCurrent^.pNext;
END_IF
END_METHOD

METHOD M_ResetPointer : BOOL
VAR_INPUT
END_VAR
pCurrent := pHead;
END_METHOD

END_PROGRAM

// ---- MainProgs/MainDispacher.TcPOU
PROGRAM MainDispacher
VAR
	fbConfig	: FB_OM_Config;
	fbInit		: FB_OM_Init;
	fbManu		: FB_OM_Manu;
	fbAuto		: FB_OM_Auto;
	fbSemiAuto	: FB_OM_SemiAuto;
	fbMaintenance : FB_OM_Maintenance;
	eForceState	: E_MachineState;
END_VAR
VAR_OUTPUT
	eCurrentMode	: E_MachineMode := E_MachineMode.MACHINEMODE_Config;
	eCurrentState	: E_MachineState;
END_VAR

CASE eCurrentMode OF
	E_MachineMode.MACHINEMODE_Config:
		fbConfig();
		eCurrentState := MAX(fbConfig.eCurrentState,eForceState);
	E_MachineMode.MACHINEMODE_Init:
		fbInit();
		eCurrentState := fbInit.eCurrentState;
	E_MachineMode.MACHINEMODE_Manu:
		fbManu();
		eCurrentState := fbManu.eCurrentState;
	E_MachineMode.MACHINEMODE_SemiAuto:
		fbSemiAuto();
		eCurrentState := fbSemiAuto.eCurrentState;
	E_MachineMode.MACHINEMODE_Auto:
		fbAuto();
		eCurrentState := fbAuto.eCurrentState;
	E_MachineMode.MACHINEMODE_Maintenance:
		fbMaintenance();
		eCurrentState := fbMaintenance.eCurrentState;
END_CASE

METHOD M_ActivateConfig : ERRORID
VAR_INPUT
END_VAR
IF eCurrentMode = E_MachineMode.MACHINEMODE_Config THEN
	M_ActivateConfig := fbConfig.M_Activate();
ELSE
	M_ActivateConfig := E_ErrorIdCmd.ERRORID_WrongMode;	//Error: nicht im Config-Modus
END_IF
END_METHOD

METHOD M_ChangeMode : ERRORID
VAR_INPUT
	eMaschineMode : E_MachineMode;
END_VAR
//Mode bereits angeforderter Mode?
IF eCurrentMode = eMaschineMode THEN
	RETURN;
END_IF

CASE eMaschineMode OF
	E_MachineMode.MACHINEMODE_Config:	
		IF eCurrentState <> E_MachineState.MACHINESTATE_Idle THEN
			M_ChangeMode := E_ErrorIdCmd.ERRORID_ModeChangeImpossible;  //Error
			RETURN;			
		END_IF
	E_MachineMode.MACHINEMODE_Init,
	E_MachineMode.MACHINEMODE_Manu,
	E_MachineMode.MACHINEMODE_SemiAuto,
	E_MachineMode.MACHINEMODE_Auto:
		IF eCurrentState <> E_MachineState.MACHINESTATE_Idle THEN
			M_ChangeMode := E_ErrorIdCmd.ERRORID_ModeChangeImpossible;  //Error
			RETURN;			
		END_IF
		IF NOT fbConfiguration.P_bActivated THEN
			M_ChangeMode := E_ErrorIdCmd.ERRORID_ConfigNotActivated;  //Error
			RETURN;
		END_IF		
	E_MachineMode.MACHINEMODE_Maintenance:
		//In Maintenance kann immer gewechselt werden
		//Der Rest wird in den enzelnen Aktionen abgefangen
		//Was ist, wenn der ActionDispacher noch aktiv ist und dann einen Fehler wirft?
		//Definitiv muss der State des ActionDispachers dann noch abgefragt werden, und dieser muss auch gestoppt werden können
		
		//Der State vom alte Mode wird übernommem
		fbMaintenance.M_SetState(eCurrentState);

		(*IF NOT (eCurrentState = E_MachineState.MACHINESTATE_Idle OR eCurrentState = E_MachineState.MACHINESTATE_Error) THEN
			M_ChangeMode := E_ErrorIdCmd.ERRORID_ModeChangeImpossible;  //Error
			RETURN;			
		END_IF*)
ELSE
	M_ChangeMode := E_ErrorIdCmd.ERRORID_UnknownMode;
	RETURN;
END_CASE

eCurrentMode := eMaschineMode;
END_METHOD

METHOD M_CheckSafety : ERRORID
VAR_INPUT
END_VAR
IF NOT (pFbSafety^.eCurrentState = E_SafetyState.Locked) THEN
	M_CheckSafety := E_ErrorIdCmd.ERRORID_InterlockNotLocked;
END_IF
END_METHOD

METHOD M_CheckSafetyInit : ERRORID
VAR_INPUT
	refData	: REFERENCE TO ARRAY[0..39] OF DINT;
END_VAR

VAR
	i : UINT;
	bInitStacker : BOOL;
	bInitOther : BOOL;
	bInitAll : BOOL;
END_VAR
bInitAll := TRUE;

FOR i := 1 TO 39 DO
	IF refData[i] > 0 THEN
		bInitAll := FALSE;
		IF fbObjectDirectory.M_GetObjType(DINT_TO_UINT(refData[i])) = E_ObjectType.OBJECTTYPE_Stacker THEN
			bInitStacker := TRUE;
		ELSE
			bInitOther := TRUE;
		END_IF
	END_IF
END_FOR

IF bInitAll THEN
	bInitOther := TRUE;
	IF fbObjectDirectory.nCntStacker > 0 THEN
		bInitStacker := TRUE;
	END_IF
END_IF

IF bInitOther THEN
	IF NOT (pFbSafety^.eCurrentState = E_SafetyState.Locked) THEN
		M_CheckSafetyInit := E_ErrorIdCmd.ERRORID_InterlockNotLocked;
	END_IF	
END_IF
END_METHOD

METHOD M_ContinueAction : ERRORID
VAR_INPUT
	nActionId	: UINT;
END_VAR
IF eCurrentState = E_MachineState.MACHINESTATE_Error THEN
	M_ContinueAction := E_ErrorIdCmd.ERRORID_InvalidState;
	RETURN;
END_IF

IF eCurrentMode = E_MachineMode.MACHINEMODE_Manu THEN
	M_ContinueAction := fbManu.M_ContinueAction(nActionId);
ELSIF eCurrentMode = E_MachineMode.MACHINEMODE_Auto THEN
	M_ContinueAction := fbAuto.M_ContinueAction(nActionId);
ELSE
	M_ContinueAction := E_ErrorIdCmd.ERRORID_WrongMode;
END_IF
END_METHOD

//Löscht die gespeicherte Konfiguration, welche nach Einschalten automatisch geladen wird
METHOD M_DeleteConfig : ERRORID
VAR_INPUT
END_VAR
IF MainDispacher.eCurrentMode = E_MachineMode.MACHINEMODE_Config THEN //im Config-Modus?
	M_DeleteConfig := fbConfig.M_Delete();
ELSE
	M_DeleteConfig := E_ErrorIdCmd.ERRORID_WrongMode;	//Error: nicht im Config-Modus
END_IF
END_METHOD

METHOD M_DeleteGCodeFiles : ERRORID
VAR_INPUT
END_VAR
END_METHOD

METHOD M_DeviceFirmwUpdate : ERRORID
VAR_INPUT
	nCanNodeId	: USINT;
END_VAR
M_DeviceFirmwUpdate := fbMaintenance.M_DeviceFirmwUpdate(nCanNodeId);
END_METHOD

METHOD M_ExeAction : ST_Error
VAR_INPUT
	eAction : E_Action;
	refData	: REFERENCE TO ARRAY[0..39] OF DINT;
END_VAR

VAR
	stActionData		: ST_ActionData;
	pDryPad				: POINTER TO FB_DryPad;
	pTipCleaner			: POINTER TO FB_TipCleaner;	
END_VAR

VAR_OUTPUT
	nActionId		: UINT;
END_VAR
IF NOT fbStopButton.P_bReleased THEN
	M_ExeAction.ErrorId := E_ErrorIdCmd.ERRORID_StopButtonNotReleased;
	eCurrentState := E_MachineState.MACHINESTATE_Error;
	RETURN;
END_IF

//Neu Action werden nur in "Idle" oder "Active" angenommen
IF NOT(eCurrentState = E_MachineState.MACHINESTATE_Idle OR
		eCurrentState = E_MachineState.MACHINESTATE_Active OR
		eCurrentState = E_MachineState.MACHINESTATE_Running OR
		eCurrentState = E_MachineState.MACHINESTATE_Pause) THEN
	M_ExeAction.ErrorId := E_ErrorIdCmd.ERRORID_WrongMode;
	RETURN;
END_IF

MEMSET(ADR(stActionData),0,SIZEOF(stActionData));
stActionData.eAction := eAction;
	
CASE eAction OF
	E_Action.ACTION_Init:
		IF eCurrentMode <> E_MachineMode.MACHINEMODE_Init THEN
			M_ExeAction.ErrorId := E_ErrorIdCmd.ERRORID_WrongMode;
			RETURN;
		END_IF
		M_ExeAction.ErrorId := M_CheckSafetyInit(refData);
	
	E_Action.ACTION_Jog,E_Action.ACTION_MoveX,E_Action.ACTION_MoveY,E_Action.ACTION_MoveXY,E_Action.ACTION_MoveZ:
		IF NOT (eCurrentMode = E_MachineMode.MACHINEMODE_Manu OR eCurrentMode = E_MachineMode.MACHINEMODE_Auto) THEN
			M_ExeAction.ErrorId := E_ErrorIdCmd.ERRORID_WrongMode;
			RETURN;			
		END_IF
		//wenn GCode aktiv, dann nur im Pause zulässig
		IF GCode.bBusy AND_THEN GCode.eGCodeState <> E_GCodeState.GCodeState_Pause THEN
			 RETURN;
		END_IF
 		
		M_ExeAction.ErrorId := M_CheckSafety();
		//BasicActions, welche nur Object und die ActionParameter benötigen 
		stActionData.nObject := DINT_TO_UINT(refData[0]);
		MEMCPY(ADR(stActionData.aParams),ADR(refData[1]),44);
	
	E_Action.ACTION_InkSpin,E_Action.ACTION_InkOpClCover,E_Action.ACTION_PowdStatReload,E_Action.ACTION_PowdStatShaking,
	E_Action.ACTION_PowdStatLeveling,E_Action.ACTION_SwitchPressure,E_Action.ACTION_PulsePressure,
	E_Action.ACTION_SwitchPump,E_Action.ACTION_OpenClose,E_Action.ACTION_LockUnlock,E_Action.ACTION_StampAdjust,
	E_Action.ACTION_Aspirate,E_Action.ACTION_Dispense,E_Action.ACTION_DispenseDrops,E_Action.ACTION_StrobTest,
	E_Action.ACTION_EmptyWaste,E_Action.ACTION_Rinse,E_Action.ACTION_Eject,E_Action.ACTION_Expose,E_Action.ACTION_Swivel,
	E_Action.ACTION_PickPutPowder,E_Action.ACTION_ReactorOpCl,E_Action.ACTION_DetectVial,E_Action.ACTION_FillLiquid,
	E_Action.ACTION_EmptyLiquid, E_Action.ACTION_StampDemolding,E_Action.ACTION_DilMoveValve,E_Action.ACTION_DilMovePlunger,
	E_Action.ACTION_DilPump, E_Action.ACTION_DilTransfer, E_Action.ACTION_SetVoltage, E_Action.ACTION_DilPrepare,
	E_Action.ACTION_SetPressure,E_Action.ACTION_SetVacuum,E_Action.ACTION_SwitchVoltage,E_Action.ACTION_Extrude,
	E_Action.ACTION_ExtrMovePlunger, E_Action.ACTION_Mix,E_Action.ACTION_MeasurepH, E_Action.ACTION_SuckOff,
	E_Action.ACTION_BasicDispense, E_Action.ACTION_StirrCartridge, E_Action.ACTION_MoveTrayTransporter, E_Action.ACTION_TurnDrivingPin,
	E_Action.ACTION_TurnTo, E_Action.ACTION_MoveLifter, E_Action.ACTION_LoadStacker:
		IF NOT (eCurrentMode = E_MachineMode.MACHINEMODE_Manu OR eCurrentMode = E_MachineMode.MACHINEMODE_Auto) THEN
			M_ExeAction.ErrorId := E_ErrorIdCmd.ERRORID_WrongMode;
			RETURN;
		END_IF
		//BasicActions, welche nur Object und die ActionParameter benötigen 
		stActionData.nObject := DINT_TO_UINT(refData[0]);
		MEMCPY(ADR(stActionData.aParams),ADR(refData[1]),44);
		
	E_Action.ACTION_WashTool, E_Action.ACTION_DryToolInside:
		IF NOT (eCurrentMode = E_MachineMode.MACHINEMODE_Manu OR eCurrentMode = E_MachineMode.MACHINEMODE_Auto) THEN
			M_ExeAction.ErrorId := E_ErrorIdCmd.ERRORID_WrongMode;
			RETURN;			
		END_IF
		M_ExeAction.ErrorId := M_CheckSafety();
		stActionData.nObject := DINT_TO_UINT(refData[0]);
		stActionData.nTarget := DINT_TO_UINT(refData[1]);
		MEMCPY(ADR(stActionData.aParams),ADR(refData[2]),60);
	
	E_Action.ACTION_MoveToTarget, E_Action.ACTION_MeasureTool, E_Action.ACTION_OpenCloseFlipTube,
	E_Action.ACTION_ExchangePiece,E_Action.ACTION_StampInking,E_Action.ACTION_CleanTip,E_Action.ACTION_DryPip,
	E_Action.ACTION_DispenseTest,E_Action.ACTION_TeachTarget,E_Action.ACTION_GetPipSample,
	E_Action.ACTION_CalibrateZSensor,E_Action.ACTION_TeachTool,E_Action.ACTION_InsertTool,E_Action.ACTION_DockTool,
	E_Action.ACTION_TransferLiquid,E_Action.ACTION_TransferGas, E_Action.ACTION_TransferTray:
		IF NOT (eCurrentMode = E_MachineMode.MACHINEMODE_Manu OR eCurrentMode = E_MachineMode.MACHINEMODE_Auto) THEN
			M_ExeAction.ErrorId := E_ErrorIdCmd.ERRORID_WrongMode;
			RETURN;			
		END_IF
		M_ExeAction.ErrorId := M_CheckSafety();
		stActionData.nObject := DINT_TO_UINT(refData[0]);
		stActionData.nTarget := DINT_TO_UINT(refData[1]);
		MEMCPY(ADR(stActionData.aParams),ADR(refData[2]),50);
	
	E_Action.ACTION_Heating,E_Action.ACTION_Cooling,E_Action.ACTION_SwitchLight:
		IF NOT (eCurrentMode = E_MachineMode.MACHINEMODE_Manu OR eCurrentMode = E_MachineMode.MACHINEMODE_Auto) THEN
			M_ExeAction.ErrorId := E_ErrorIdCmd.ERRORID_WrongMode;
			RETURN;			
		END_IF
		stActionData.nObject := DINT_TO_UINT(refData[0]);
		MEMCPY(ADR(stActionData.aParams),ADR(refData[1]),16);
	
	E_Action.ACTION_Delay:
		MEMCPY(ADR(stActionData.aParams),ADR(refData[0]),4);

	E_Action.ACTION_ActionOnArray:
		IF eCurrentMode <> E_MachineMode.MACHINEMODE_Manu THEN
			M_ExeAction.ErrorId := E_ErrorIdCmd.ERRORID_WrongMode;
			RETURN;			
		END_IF
		M_ExeAction.ErrorId := M_CheckSafety();
		stActionData.nObject := DINT_TO_UINT(refData[0]);
		stActionData.nTarget := DINT_TO_UINT(refData[1]);
		MEMCPY(ADR(stActionData.aParams),ADR(refData[2]),72);
	
	E_Action.ACTION_ChangeCleanMat:
		stActionData.nObject := DINT_TO_UINT(refData[0]);
		IF fbObjectDirectory.M_GetObjType(stActionData.nObject) = E_ObjectType.OBJECTTYPE_DryPad THEN
			pDryPad := fbObjectDirectory.M_GetObjPointer(stActionData.nObject);
			pDryPad^.M_ChangeCleanMat();
			RETURN;
		ELSIF fbObjectDirectory.M_GetObjType(stActionData.nObject) = E_ObjectType.OBJECTTYPE_TipCleaner THEN
			pTipCleaner := fbObjectDirectory.M_GetObjPointer(stActionData.nObject);
			pTipCleaner^.M_ChangeCleanMat();
			RETURN;
		ELSE
			M_ExeAction.ErrorId := E_ErrorIdCmd.ERRORID_UnsuitableObject;
		END_IF
	E_Action.ACTION_RunGCode:
		IF eCurrentMode <> E_MachineMode.MACHINEMODE_Manu THEN
			M_ExeAction.ErrorId := E_ErrorIdCmd.ERRORID_WrongMode;
			RETURN;			
		END_IF
		stActionData.nTarget := DINT_TO_UINT(refData[0]);
		MEMCPY(ADR(stActionData.aParams),ADR(refData[1]),48);
	E_Action.ACTION_RunSequence:
		IF eCurrentMode <> E_MachineMode.MACHINEMODE_Auto THEN
			M_ExeAction.ErrorId := E_ErrorIdCmd.ERRORID_WrongMode;
			RETURN;			
		END_IF
		MEMCPY(ADR(stActionData.aParams),ADR(refData[0]),24);
	E_Action.ACTION_ShiftGCodeZPos:
		MEMCPY(ADR(stActionData.aParams),ADR(refData[0]),4);
	E_Action.ACTION_MoveAllHome:
		IF NOT (eCurrentMode = E_MachineMode.MACHINEMODE_Manu OR eCurrentMode = E_MachineMode.MACHINEMODE_Auto) THEN
			M_ExeAction.ErrorId := E_ErrorIdCmd.ERRORID_WrongMode;
			RETURN;
		ELSE
			IF eCurrentState <> E_MachineState.MACHINESTATE_Idle THEN
				M_ExeAction.ErrorId := E_ErrorIdCmd.ERRORID_InvalidState;
				RETURN;
			END_IF
		END_IF
	E_Action.ACTION_CoupleHeads:
		IF eCurrentState <> E_MachineState.MACHINESTATE_Idle THEN
			M_ExeAction.ErrorId := E_ErrorIdCmd.ERRORID_InvalidState;
			RETURN;
		END_IF
		MEMCPY(ADR(stActionData.aParams),ADR(refData[0]),4);
ELSE
	M_ExeAction.ErrorId := E_ErrorIdCmd.ERRORID_InvalidAction;
END_CASE

IF M_ExeAction.ErrorId > 0 THEN
	RETURN;
END_IF

CASE eCurrentMode OF
	E_MachineMode.MACHINEMODE_Init:
		M_ExeAction := fbInit.M_ExeAction(refData);
	E_MachineMode.MACHINEMODE_Manu:
		M_ExeAction.ErrorId := fbManu.M_ExeAction(refActionData:= stActionData,nActionId=> nActionId);
	E_MachineMode.MACHINEMODE_Auto:
		M_ExeAction.ErrorId := fbAuto.M_ExeAction(refActionData:= stActionData,nActionId=> nActionId);
	//Hier könnte gecheckt werden, in welchem Mode eine Action ausgeführt werden kann (Pause oder so)
	;
END_CASE
END_METHOD

METHOD M_ForceError
VAR_INPUT
END_VAR
eCurrentState := E_MachineState.MACHINESTATE_Error;
eForceState := E_MachineState.MACHINESTATE_Error;
END_METHOD

METHOD M_PauseAction : ERRORID
VAR_INPUT
	nActionId	: UINT;
END_VAR
IF eCurrentState = E_MachineState.MACHINESTATE_Error THEN
	M_PauseAction := E_ErrorIdCmd.ERRORID_InvalidState;
	RETURN;
END_IF

IF eCurrentMode = E_MachineMode.MACHINEMODE_Manu THEN
	fbManu.M_PauseAction(nActionId);
ELSIF eCurrentMode = E_MachineMode.MACHINEMODE_Auto THEN
	fbAuto.M_PauseAction(nActionId);
END_IF
END_METHOD

METHOD M_ResetError
VAR_INPUT
END_VAR
fbConfig.M_ResetError();
fbInit.M_ResetError();
fbManu.M_ResetError();
fbSemiAuto.M_ResetError();
fbAuto.M_ResetError();
fbMaintenance.M_ResetError();
//GCode.M_Reset();
eCurrentState := E_MachineState.MACHINESTATE_Reset;
END_METHOD

METHOD M_ResetPlc : ERRORID
VAR_INPUT
END_VAR
M_ChangeMode(E_MachineMode.MACHINEMODE_Maintenance);
M_ResetPlc := fbMaintenance.M_ResetPlc();
END_METHOD

METHOD M_SaveConfig : ERRORID
VAR_INPUT
END_VAR
IF eCurrentMode = E_MachineMode.MACHINEMODE_Config THEN //im Config-Modus?
	M_SaveConfig := fbConfig.M_Save();
ELSE
	M_SaveConfig := E_ErrorIdCmd.ERRORID_WrongMode;	//Error: nicht im Config-Modus
END_IF
END_METHOD

METHOD M_SetupAxis : ERRORID
VAR_INPUT
	refCmdData : REFERENCE TO ST_CmdData;
END_VAR
IF eCurrentMode = E_MachineMode.MACHINEMODE_Maintenance THEN
	M_SetupAxis := fbMaintenance.M_SetupAxis(refCmdData);
ELSE
	M_SetupAxis := E_ErrorIdCmd.ERRORID_WrongMode;
END_IF
END_METHOD

METHOD M_StopAction : ERRORID
VAR_INPUT
	nActionId	: UINT;
END_VAR
IF eCurrentState = E_MachineState.MACHINESTATE_Error THEN
	M_StopAction := E_ErrorIdCmd.ERRORID_InvalidState;
	RETURN;
END_IF

IF eCurrentMode = E_MachineMode.MACHINEMODE_Manu THEN
	M_StopAction := fbManu.M_StopAction(nActionId);
ELSIF eCurrentMode = E_MachineMode.MACHINEMODE_Auto THEN
	M_StopAction := fbAuto.M_StopAction(nActionId);
ELSE
	M_StopAction := E_ErrorIdCmd.ERRORID_WrongMode;
END_IF
END_METHOD

METHOD M_StopAll
VAR_INPUT
END_VAR
IF eCurrentMode = E_MachineMode.MACHINEMODE_Init THEN
	fbInit.M_Cancel();	
ELSIF eCurrentMode = E_MachineMode.MACHINEMODE_Manu THEN
	fbManu.M_Cancel();
ELSIF eCurrentMode = E_MachineMode.MACHINEMODE_Auto THEN
	fbAuto.M_Cancel();
ELSIF eCurrentMode = E_MachineMode.MACHINEMODE_Maintenance THEN
	fbMaintenance.M_Cancel();
END_IF
END_METHOD

PROPERTY P_bReadyToUnlock : BOOL
GET
IF eCurrentMode = E_MachineMode.MACHINEMODE_Config THEN
	P_bReadyToUnlock := TRUE;
ELSE
	IF eCurrentState = E_MachineState.MACHINESTATE_Idle OR eCurrentState = E_MachineState.MACHINESTATE_Error THEN
		P_bReadyToUnlock := TRUE;	
	END_IF
END_IF
END_GET
END_PROPERTY

PROPERTY P_eCurrentState : E_MachineState
GET
CASE eCurrentMode OF
	E_MachineMode.MACHINEMODE_Config:
		P_eCurrentState := fbConfig.eCurrentState;
	E_MachineMode.MACHINEMODE_Init:
		P_eCurrentState := fbInit.eCurrentState;
	E_MachineMode.MACHINEMODE_Manu:
		P_eCurrentState := fbManu.eCurrentState;
	E_MachineMode.MACHINEMODE_SemiAuto:
		P_eCurrentState := fbSemiAuto.eCurrentState;
	E_MachineMode.MACHINEMODE_Auto:
		P_eCurrentState := fbAuto.eCurrentState;
	E_MachineMode.MACHINEMODE_Maintenance:
		P_eCurrentState := fbMaintenance.eCurrentState;
END_CASE
END_GET
END_PROPERTY

END_PROGRAM

// ---- OperatingModes/FB_OM_Config.TcPOU
FUNCTION_BLOCK FB_OM_Config
VAR_INPUT
END_VAR
VAR_OUTPUT
	eCurrentState : E_MachineState := E_MachineState.MACHINESTATE_Idle;
END_VAR
VAR
	bFirstCycle				: BOOL := TRUE;
	stError					: ST_Error;
	bError					: BOOL;
	bBusy					: BOOL;
	
	//ConfigActions
	nStateA_ConfigAction	: USINT;
	bActivate				: BOOL;
	nActivateCnt1			: USINT; //allg Zählvariable
	
	bSaveCurrConfig			: BOOL;
	bLoadConfig				: BOOL;
	bDeleteConfig			: BOOL;
	
	nStateA_CheckObjProps	: USINT;
	iter					: FB_ObjCollectIteratorDeep;
	pObject					: POINTER TO FB_Object;
	nCheckObjCounter		: USINT;
	
	nStateA_Reset			: USINT;
	i						: UINT;
	bSetupDefaultObjOk		: BOOL;
	timer					: TON;
	
	bWriteXYAxisPara		: BOOL;
	nStateA_WriteXYAxisPara	: USINT;
	
	bSimError				: BOOL;
END_VAR

IF bFirstCycle THEN
	bFirstCycle := FALSE;
	bLoadConfig := fbConfiguration.P_bConfigSaved;
	eCurrentState := E_MachineState.MACHINESTATE_Active;	
END_IF

IF eCurrentState = E_MachineState.MACHINESTATE_Active THEN
	IF bLoadConfig THEN
		fbConfiguration.A_Load(bExecute:= TRUE);
		IF NOT fbConfiguration.bBusy THEN
			IF fbConfiguration.bError THEN
				bError := TRUE;
				fbErrorList.M_Add(stError);
			ELSE
				bActivate := TRUE;
			END_IF
			fbConfiguration.A_Load(bExecute:= FALSE);
			bLoadConfig := FALSE;
			//bei erfolg Konfiguration laden
		END_IF
	ELSIF bDeleteConfig THEN
		fbConfiguration.A_Delete(bExecute:= TRUE);
		IF NOT fbConfiguration.bBusy THEN
			IF fbConfiguration.bError THEN
				bError := TRUE;
				fbErrorList.M_Add(stError);
			END_IF
			fbConfiguration.A_Delete(bExecute:= FALSE);
			bDeleteConfig := FALSE;
		END_IF
	ELSIF bActivate THEN	//Konfiguration aktivieren
		fbConfiguration.A_Activate(bExecute:= TRUE);
		IF NOT fbConfiguration.bBusy THEN
			IF fbConfiguration.bError THEN
				bError := TRUE;
				fbErrorList.M_Add(fbConfiguration.stError);
			END_IF
			fbConfiguration.A_Activate(bExecute:= FALSE);
			bActivate := FALSE;
		END_IF
	ELSIF bSaveCurrConfig THEN
		fbConfiguration.A_Save(bExecute:= TRUE);
		IF NOT fbConfiguration.bBusy THEN
			IF fbConfiguration.bError THEN
				bError := TRUE;
				fbErrorList.M_Add(stError);
			END_IF
			fbConfiguration.A_Save(bExecute:= FALSE);
			bSaveCurrConfig := FALSE;
		END_IF
	END_IF

	IF NOT (bActivate OR bSaveCurrConfig OR bLoadConfig OR bDeleteConfig) THEN
		IF bError THEN
			eCurrentState := E_MachineState.MACHINESTATE_Error;
		ELSE
			eCurrentState := E_MachineState.MACHINESTATE_Idle;
		END_IF
	END_IF
	
ELSIF eCurrentState = E_MachineState.MACHINESTATE_Reset THEN
	A_Reset();
	IF nStateA_Reset = 80 THEN
		nStateA_Reset := 0;
		bError := FALSE;
		eCurrentState := E_MachineState.MACHINESTATE_Idle;
	ELSIF nStateA_Reset = 99 THEN
		nStateA_Reset := 0;
		eCurrentState := E_MachineState.MACHINESTATE_Error;
	END_IF
ELSIF eCurrentState = E_MachineState.MACHINESTATE_Idle THEN
	//Auf Fehler der Hardware reagieren
	IF PerformHardware.bError THEN
		eCurrentState := E_MachineState.MACHINESTATE_Error;
	END_IF
END_IF

IF bSimError THEN
	eCurrentState := E_MachineState.MACHINESTATE_Error;
END_IF

METHOD M_Delete : ERRORID
VAR_INPUT
END_VAR
IF eCurrentState = E_MachineState.MACHINESTATE_Idle THEN
	bDeleteConfig := TRUE;
	eCurrentState := E_MachineState.MACHINESTATE_Active;
END_IF
END_METHOD

METHOD M_Activate : ERRORID
VAR_INPUT
END_VAR
IF eCurrentState = E_MachineState.MACHINESTATE_Idle THEN
	bActivate := TRUE;
	eCurrentState := E_MachineState.MACHINESTATE_Active;
ELSE
	M_Activate := E_ErrorIdCmd.ERRORID_InvalidState;
END_IF
END_METHOD

METHOD M_ResetError
VAR_INPUT
END_VAR
IF eCurrentState = E_MachineState.MACHINESTATE_Error THEN
	eCurrentState := E_MachineState.MACHINESTATE_Reset;
	bError := FALSE;
END_IF
END_METHOD

METHOD M_Save : ERRORID
VAR_INPUT
END_VAR
IF eCurrentState = E_MachineState.MACHINESTATE_Idle THEN
	bSaveCurrConfig := TRUE;
	eCurrentState := E_MachineState.MACHINESTATE_Active;
ELSE
	M_Save := E_ErrorIdCmd.ERRORID_InvalidState;
END_IF
END_METHOD

ACTION A_Reset:
//In Config gehen die Objekte selber nicht in Error, da an diesen keine Actions ausgeführt werden
//Es kann also nur die Hardware in Error gehen, folglich braucht auch nur dieses zurückgesetzt werden
IF nStateA_Reset = 0 THEN
	IF PerformHardware.bError THEN
		PerformHardware.A_ResetError();
		timer(IN:= TRUE, PT:=T#20S);
		IF timer.Q THEN
			timer(IN:= FALSE);
			nStateA_Reset := 99;
		END_IF
	ELSE
		timer(IN:= FALSE);
		nStateA_Reset := 80;
	END_IF	
END_IF
END_ACTION

ACTION A_CheckObjProps:
IF nStateA_CheckObjProps = 0 THEN
	nCheckObjCounter := 0;
	fbObjectDirectory.P_pDeviceCollection^.M_GetIterator(iter);
	nStateA_CheckObjProps := 1;
END_IF

WHILE iter.pNode > 0 AND_THEN iter.pNode^.P_pObject > 0 DO
	pObject := iter.pNode^.P_pObject;
	nCheckObjCounter := nCheckObjCounter + 1;
	stError.ObjectId := pObject^.P_nObjectID;
	stError.ErrorId := pObject^.M_CheckProps();
	IF stError.ErrorId > 0 THEN
		nStateA_CheckObjProps := 99;
		RETURN;
	END_IF
	iter.M_Increment();
	IF nCheckObjCounter = 100 THEN
		nCheckObjCounter := 0;
		RETURN;
	END_IF
END_WHILE

nStateA_CheckObjProps := 80;
END_ACTION

END_FUNCTION_BLOCK

// ---- Hardware/PerformHardware.TcPOU
PROGRAM PerformHardware
VAR
	i : UINT;
	nIndex : USINT;
	nHwDataIndex : USINT;
	stHardwareId : ST_HardwareId;
	pHwModule : POINTER TO FB_HwModule;
END_VAR
VAR_OUTPUT
	bError : BOOL;
END_VAR

bError := FALSE;

nHwDataIndex := 0;

fbPCV();

fbStopButton();
IF fbStopButton.P_bTriggered THEN
	MainDispacher.M_StopAll();
	{IF defined (variable:fbHighVoltSupplyRef)}
	fbHighVoltSupplyRef.M_SwitchVoltage(1, FALSE);
	fbHighVoltSupplyRef.M_SwitchVoltage(2, FALSE);
	{END_IF}
END_IF

pFbSafety^();
IF pFbSafety^.eCurrentState <> E_SafetyState.Locked THEN
	MainDispacher.M_StopAll();
END_IF

//HardwareId bilden (Safety)
stHardwareId.eGroup := E_HardwareGrp.Interlock;
stHardwareId.nParentItem := 0;
stHardwareId.nItem := 1;
MEMCPY(ADR(aHardwProcData[nHwDataIndex].nHardwareId),ADR(stHardwareId),4);

aHardwProcData[nHwDataIndex].nInterpretation := 0;
aHardwProcData[nHwDataIndex].nValue := pFbSafety^.eCurrentState;
nHwDataIndex := nHwDataIndex + 1;

{IF defined(variable:fbSafetyStacker)}
fbSafetyStacker();
stHardwareId.eGroup := E_HardwareGrp.Interlock;
stHardwareId.nParentItem := 0;
stHardwareId.nItem := 2;
MEMCPY(ADR(aHardwProcData[nHwDataIndex].nHardwareId),ADR(stHardwareId),4);

aHardwProcData[nHwDataIndex].nInterpretation := 0;
aHardwProcData[nHwDataIndex].nValue := fbSafetyStacker.eCurrentState;
nHwDataIndex := nHwDataIndex + 1;
{END_IF}

fbXYDriveList.M_SetCurrentToHead();
REPEAT
	pHwModule := fbXYDriveList.M_Get();
	IF pHwModule > 0 THEN
		pHwModule^();
		IF pHwModule^.P_bError THEN
			bError := TRUE;
		END_IF
	END_IF
UNTIL pHwModule = 0
END_REPEAT

fbCANOpenHwModuleList.M_SetCurrentToHead();
REPEAT
	pHwModule := fbCANOpenHwModuleList.M_Get();
	IF pHwModule > 0 THEN
		pHwModule^();
		IF pHwModule^.P_bError THEN
			bError := TRUE;	
		END_IF
	END_IF
UNTIL pHwModule = 0
END_REPEAT

FOR i:= 1 TO cNoOfGearPumps BY 1 DO
	aFbGearPumps[i]();
END_FOR

//Ampel für Printer allgemein
fbSignalLight(eSafetyState:= fbSafety.eCurrentState, eMachineState:= MainDispacher.eCurrentState);	
//Ampel für Stacker
{IF defined(Stacker)}
fbSignalLightStacker(eSafetyState:= fbSafetyStacker.eCurrentState, eMachineState:= afbStacker[1].P_eCurrentState);
{END_IF}

fbMultiZDigiOut();
fbPlcTriggerOut();
fbMultiZPWM();

{IF defined(variable:fbHighVoltSupplyRef)}
fbHighVoltSupplyRef();
{END_IF}

{IF defined(variable:fbUnistatRef)}
fbUnistatRef();
{END_IF}

{IF defined(variable:fbHwRefTrayLock)}
fbHwRefTrayLock();
{END_IF}

{IF defined(variable:fbHwRefSpinDrive)}
fbHwRefSpinDrive();
{END_IF}

{IF defined(variable:fbHwRefLiftDrive)}
fbHwRefLiftDrive();
{END_IF}

{IF defined(variable:fbHwRefTrayStop)}
fbHwRefTrayStop();
{END_IF}

//Aktuelle Werte PneuChannels für GUI (wird in aktueller GUI nicht ausgewertet)
stHardwareId.eGroup := E_HardwareGrp.PneuChannel;
stHardwareId.nParentItem := 0;
FOR i:= 0 TO cNoOfPneuChannels - 1 BY 1 DO
	nIndex := UINT_TO_USINT(i + 1);
	stHardwareId.nItem := nIndex;
	aFbPneuChannel[nIndex]();
	MEMCPY(ADR(aHardwProcData[nHwDataIndex].nHardwareId),ADR(stHardwareId),4);	
	aHardwProcData[nHwDataIndex].nInterpretation := 0;
	aHardwProcData[nHwDataIndex].nValue := BOOL_TO_DINT(aFbPneuChannel[nIndex].P_bSupplyOk);
	nHwDataIndex := nHwDataIndex + 1;
	MEMCPY(ADR(aHardwProcData[nHwDataIndex].nHardwareId),ADR(stHardwareId),4);
	aHardwProcData[nHwDataIndex].nInterpretation := 1;
	aHardwProcData[nHwDataIndex].nValue := aFbPneuChannel[nIndex].P_nSetPressure;
	nHwDataIndex := nHwDataIndex + 1;
	MEMCPY(ADR(aHardwProcData[nHwDataIndex].nHardwareId),ADR(stHardwareId),4);	
	aHardwProcData[nHwDataIndex].nInterpretation := 2;
	aHardwProcData[nHwDataIndex].nValue := aFbPneuChannel[nIndex].P_nCurrentPressure;
	nHwDataIndex := nHwDataIndex + 1;
END_FOR

ACTION A_ResetError:
fbXYDriveList.M_SetCurrentToHead();
REPEAT
	pHwModule := fbXYDriveList.M_Get();
	IF pHwModule > 0 THEN
		pHwModule^.M_Reset();
	END_IF
UNTIL pHwModule = 0
END_REPEAT

fbCANOpenHwModuleList.M_SetCurrentToHead();
REPEAT
	pHwModule := fbCANOpenHwModuleList.M_Get();
	IF pHwModule > 0 THEN
		pHwModule^.M_Reset();
	END_IF
UNTIL pHwModule = 0
END_REPEAT
END_ACTION

END_PROGRAM

// ---- OperatingModes/FB_OM_Init.TcPOU
FUNCTION_BLOCK FB_OM_Init
VAR_INPUT
END_VAR
VAR_OUTPUT
	eCurrentState : E_MachineState := E_MachineState.MACHINESTATE_Idle;
END_VAR
VAR
	stActionData 	: ST_ActionData := (eAction := E_Action.ACTION_Init);
	i				: UINT;	
	stError 		: ST_Error;
	nStateA_Reset 	: USINT;
	timeout 		: TON;	
END_VAR

CASE eCurrentState OF
	E_MachineState.MACHINESTATE_Idle:
		//Auf Fehler der Hardware reagieren
		IF PerformHardware.bError THEN
			eCurrentState := E_MachineState.MACHINESTATE_Error;
		END_IF
	E_MachineState.MACHINESTATE_Active:
		eCurrentState := ActionDispacher.eCurrentState;
	E_MachineState.MACHINESTATE_Cancel:
		ActionDispacher.M_StopAll();
		eCurrentState := ActionDispacher.eCurrentState;
	E_MachineState.MACHINESTATE_Canceled:
		eCurrentState := ActionDispacher.eCurrentState;
	E_MachineState.MACHINESTATE_Reset:
		A_Reset();
	E_MachineState.MACHINESTATE_Error:
		//Do Nothing		
END_CASE

ACTION A_Reset:
IF nStateA_Reset = 0 THEN
	//ActionDispacher zurücksetzen (Hier werden auch die Devices zurückgesetzt
	ActionDispacher.M_Reset();
	//Hardware zurücksetzen
	PerformHardware.A_ResetError();
	//PCV zurücksetzen
	timeout(IN:= FALSE);
	nStateA_Reset := 1;
ELSIF nStateA_Reset = 1 THEN
	nStateA_Reset := 2;
	timeout(IN:= TRUE, PT:=T#20S);
	//Warten, bis alles zurückgesetzt
	IF ActionDispacher.eCurrentState <> E_MachineState.MACHINESTATE_Idle THEN
		nStateA_Reset := 1; 		
	END_IF
	IF PerformHardware.bError THEN
		PerformHardware.A_ResetError();
		nStateA_Reset := 1;
	END_IF
	IF timeout.Q THEN
		eCurrentState := E_MachineState.MACHINESTATE_Error;
		nStateA_Reset := 0;
	END_IF
ELSIF nStateA_Reset = 2 THEN
	//Checken, ob MzBase komplett resettet wurde -> Aktivierung der KOnfiguration erforderlich
	FOR i:= 1 TO cMaxMzHeads BY 1 DO
		IF aFbMultiZRef[i].P_bMzBaseRestarted THEN
			fbConfiguration.M_Deactivate();
		END_IF
	END_FOR
	
	IF fbConfiguration.P_bActivated THEN
		eCurrentState := E_MachineState.MACHINESTATE_Idle;
		nStateA_Reset := 0;
	ELSE
		nStateA_Reset := 3;
	END_IF
ELSIF nStateA_Reset = 3 THEN //Konfiguration wieder aktivieren
	fbConfiguration.A_Activate(bExecute:= TRUE);
	IF NOT fbConfiguration.bBusy THEN
		IF fbConfiguration.bError THEN
			eCurrentState := E_MachineState.MACHINESTATE_Error;
			fbErrorList.M_Add(stError);
		ELSE
			eCurrentState := E_MachineState.MACHINESTATE_Idle;
		END_IF
		nStateA_Reset := 0;
		fbConfiguration.A_Activate(bExecute:= FALSE);
	END_IF
END_IF
END_ACTION

METHOD M_Cancel : ERRORID
VAR_INPUT
END_VAR
VAR
END_VAR
IF eCurrentState = E_MachineState.MACHINESTATE_Active THEN	//auf Cancel-Kommando braucht nur im Actice-State reagiert werden
	ActionDispacher.M_StopAll();
END_IF
END_METHOD

METHOD M_ExeAction : ST_Error
VAR_INPUT
	refData : REFERENCE TO ARRAY[0..39] OF DINT;
END_VAR

VAR
	i				: UINT;
	bInitAllObjects : BOOL;
	iter			: FB_ObjCollectIterator;
END_VAR
M_ExeAction.Cmd := E_Action.ACTION_Init;

//Start der Initialisierung nur in "Idle" möglich
IF NOT (eCurrentState = E_MachineState.MACHINESTATE_Idle) THEN
	M_ExeAction.ErrorId := E_ErrorIdCmd.ERRORID_InvalidState;
	RETURN;
ELSE
	
	stActionData.aParams[1] := refData[0];
	
	IF NOT stActionData.eAction = E_Action.ACTION_Init THEN
		RETURN;
	END_IF
	
	bInitAllObjects := TRUE;
	
	FOR i:= 1 TO 39 BY 1 DO
		IF refData[i] > 0 THEN
			IF refData[i] <= fbObjectDirectory.nCntObject THEN	//gültiges Object?
				IF NOT fbObjectDirectory.M_ObjIsDevice(DINT_TO_UINT(refData[i])) THEN
					M_ExeAction.ObjectId := DINT_TO_UINT(refData[i]);
					M_ExeAction.ErrorId := E_ErrorIdObjMgmt.ERRORID_IsNoDevice;	//Error: Object ist kein Device			
				END_IF
			ELSE
				M_ExeAction.ObjectId := DINT_TO_UINT(refData[i]);
				M_ExeAction.ErrorId := E_ErrorIdCmd.ERRORID_ObjectNotExists;	//Error: Object existiert nicht
				RETURN;
			END_IF
			bInitAllObjects := FALSE;
		END_IF
	END_FOR
	
	IF bInitAllObjects THEN	//Alle Devices initialisieren
		fbObjectDirectory.P_pDeviceCollection^.M_GetIterator(iter);
		WHILE iter.pNode > 0 AND_THEN iter.pNode^.P_pObject > 0 DO
			//Falls ein Diluter initialisiert wird, muss das eventuell vorhandene Pneumatikventil am PCV ausgeschalten werden
			//Das Pneumatikventil existiert nur bei Versionen mit SolenoidPip,welche zum Dispensen Druck über das PCV bezieht
				IF iter.pNode^.P_pObject^.P_eObjectType = E_ObjectType.OBJECTTYPE_Diluter THEN
				fbPCV.M_SwitchPneuValve(FALSE);
			END_IF
			stActionData.nObject := iter.pNode^.P_pObject^.P_nObjectID;
			M_ExeAction.ObjectId := iter.pNode^.P_pObject^.P_nObjectID;
			M_ExeAction.ErrorId := ActionDispacher.M_ExeAction(stActionData, TRUE);
			IF M_ExeAction.ErrorId > 0 THEN
				RETURN;
			END_IF				
			iter.M_Increment();
		END_WHILE
	ELSE	//nur in "aObjectId" angegebene Devices initialisieren
		FOR i:= 1 TO 39 BY 1 DO
			IF refData[i] > 0 THEN
				//Falls ein Diluter initialisiert wird, muss das eventuell vorhandene Pneumatikventil am PCV ausgeschalten werden
				//Das Pneumatikventil existiert nur bei Versionen mit SolenoidPip,welche zum Dispensen Druck über das PCV bezieht
				stActionData.nObject := DINT_TO_UINT(refData[i]);
				IF fbObjectDirectory.M_GetObjType(stActionData.nObject) = E_ObjectType.OBJECTTYPE_Diluter THEN
					fbPCV.M_SwitchPneuValve(FALSE);
				END_IF
				M_ExeAction.ObjectId := stActionData.nObject;
				M_ExeAction.ErrorId := ActionDispacher.M_ExeAction(stActionData, TRUE);
				IF M_ExeAction.ErrorId > 0 THEN
					RETURN;
				END_IF				
			END_IF
		END_FOR
	END_IF
	eCurrentState := E_MachineState.MACHINESTATE_Active;
END_IF
END_METHOD

METHOD M_ResetError
VAR_INPUT
END_VAR
IF eCurrentState = E_MachineState.MACHINESTATE_Error THEN 
	eCurrentState := E_MachineState.MACHINESTATE_Reset;
END_IF
END_METHOD

END_FUNCTION_BLOCK

// ---- OperatingModes/FB_OM_Manu.TcPOU
FUNCTION_BLOCK FB_OM_Manu

VAR_OUTPUT
	eCurrentState : E_MachineState := E_MachineState.MACHINESTATE_Idle;
END_VAR

VAR
	i : UINT;
	stError : ST_Error;
	nStateA_Reset : USINT;
	timeout : TON;
END_VAR

CASE eCurrentState OF
	E_MachineState.MACHINESTATE_Idle:
		A_FillPCV();
		//Auf Fehler der Hardware reagieren und eventuelle CustomUnitType2 reagieren
		IF PerformHardware.bError OR fbObjectDirectory.M_CustomUnitType2_Error() THEN
			eCurrentState := E_MachineState.MACHINESTATE_Error;
		END_IF
		
	E_MachineState.MACHINESTATE_Active:
		A_FillPCV();
		eCurrentState := ActionDispacher.eCurrentState;
		IF fbObjectDirectory.M_CustomUnitType2_Error() THEN
			ActionDispacher.M_StopAll();
			eCurrentState := E_MachineState.MACHINESTATE_Error;
		END_IF
	E_MachineState.MACHINESTATE_Cancel:
		ActionDispacher.M_StopAll();
		eCurrentState := ActionDispacher.eCurrentState;
	E_MachineState.MACHINESTATE_Canceled:
		eCurrentState := ActionDispacher.eCurrentState;
	E_MachineState.MACHINESTATE_Reset:
		A_Reset();
	E_MachineState.MACHINESTATE_Error:
		//Do nothing
END_CASE

ACTION A_FillPCV:
IF (fbObjectDirectory.nCntPiezoPip > 0) OR (fbObjectDirectory.nCntSolenoidPip > 0) THEN
	fbPCV.M_Fill();
	IF fbPCV.bError THEN
		stError.HardwareGrp := E_HardwareGrp.PCV;
		stError.HardwareNr := 1;
		stError.MachineMode := E_MachineMode.MACHINEMODE_Manu;
		stError.POU := 1;
		stError.POUAction := E_POUACT.POUACT_UNDEFIEND;
		stError.ErrorId := fbPCV.nErrorId;
		fbErrorList.A_Add(putValue := stError);
		ActionDispacher.M_StopAll();
		eCurrentState := E_MachineState.MACHINESTATE_Error;
		RETURN;
	END_IF
END_IF
END_ACTION

ACTION A_Reset:
IF nStateA_Reset = 0 THEN
	//ActionDispacher zurücksetzen (Hier werden auch die Devices zurückgesetzt)
	ActionDispacher.M_Reset();
	//Hardware zurücksetzen
	PerformHardware.A_ResetError();
	//PCV zurücksetzen
	fbPCV.M_Reset();
	timeout(IN:= FALSE);
	nStateA_Reset := 1;
ELSIF nStateA_Reset = 1 THEN
	nStateA_Reset := 2;
	timeout(IN:= TRUE, PT:=T#20S);
	//Warten, bis alles zurückgesetzt
	IF ActionDispacher.eCurrentState <> E_MachineState.MACHINESTATE_Idle THEN
		nStateA_Reset := 1; 		
	END_IF
	IF PerformHardware.bError THEN
		PerformHardware.A_ResetError();
		nStateA_Reset := 1;
	END_IF
	IF timeout.Q THEN
		eCurrentState := E_MachineState.MACHINESTATE_Error;
		nStateA_Reset := 0;
	END_IF
ELSIF nStateA_Reset = 2 THEN
	//Reset CustomUnitType2 (kann möglicherweise noch in Error stehen, weil evtl. ActionDispacher nicht in Error war)
	//Dadurch werden Objekte diesen Typs nicht durch den AD zurückgesetzt.
	fbObjectDirectory.M_ResetCustomUnitType2();
	
	//Checken, ob MzBase komplett resettet wurde -> Aktivierung der Konfiguration erforderlich
	FOR i:= 1 TO cMaxMzHeads BY 1 DO
		IF aFbMultiZRef[i].P_bMzBaseRestarted THEN
			fbConfiguration.M_Deactivate();
		END_IF
	END_FOR
	
	IF fbConfiguration.P_bActivated THEN
		eCurrentState := E_MachineState.MACHINESTATE_Idle;
		nStateA_Reset := 0;
	ELSE
		nStateA_Reset := 3;
	END_IF
ELSIF nStateA_Reset = 3 THEN //Konfiguration wieder aktivieren
	fbConfiguration.A_Activate(bExecute:= TRUE);
	IF NOT fbConfiguration.bBusy THEN
		IF fbConfiguration.bError THEN
			eCurrentState := E_MachineState.MACHINESTATE_Error;
			fbErrorList.M_Add(stError);
		ELSE
			eCurrentState := E_MachineState.MACHINESTATE_Idle;
		END_IF
		nStateA_Reset := 0;
		fbConfiguration.A_Activate(bExecute:= FALSE);
	END_IF
END_IF
END_ACTION

METHOD M_Cancel : ERRORID
VAR_INPUT
END_VAR
VAR
END_VAR
IF eCurrentState = E_MachineState.MACHINESTATE_Active THEN	//auf Cancel-Kommando braucht nur im Actice-State reagiert werden
	ActionDispacher.M_StopAll();
END_IF
END_METHOD

METHOD M_ContinueAction : ERRORID
VAR_INPUT
	nActionId	: UINT;
END_VAR
IF ActionDispacher.eCurrentState = E_MachineState.MACHINESTATE_Active THEN
	M_ContinueAction := ActionDispacher.M_ContinueAction(nActionId);
END_IF
END_METHOD

METHOD M_ExeAction : ERRORID
VAR_INPUT
	refActionData	: REFERENCE TO ST_ActionData;
END_VAR

VAR_OUTPUT
	nActionId		: UINT;
END_VAR

VAR
	nErrorId		: ERRORID;
END_VAR
//Manuelle Kommandos nur in "Idle" und "Active" möglich
IF NOT ((eCurrentState = E_MachineState.MACHINESTATE_Idle) OR (eCurrentState = E_MachineState.MACHINESTATE_Active) ) THEN
	M_ExeAction := E_ErrorIdCmd.ERRORID_InvalidState;
	RETURN;
ELSE
	nErrorId := ActionDispacher.M_ExeAction(refActionData:= refActionData, bExtern:= TRUE, nActionId=> nActionId);
	IF nErrorId > 0 THEN
		M_ExeAction := nErrorId;
		RETURN;
	ELSE
		eCurrentState := E_MachineState.MACHINESTATE_Active;
	END_IF
END_IF
END_METHOD

METHOD M_PauseAction : ERRORID
VAR_INPUT
	nActionId	: UINT;
END_VAR
IF ActionDispacher.eCurrentState = E_MachineState.MACHINESTATE_Active THEN
	M_PauseAction := ActionDispacher.M_PauseAction(nActionId);
END_IF
END_METHOD

METHOD M_ResetError
VAR_INPUT
END_VAR
IF eCurrentState = E_MachineState.MACHINESTATE_Error THEN
	eCurrentState := E_MachineState.MACHINESTATE_Reset;
END_IF
END_METHOD

METHOD M_StopAction : ERRORID
VAR_INPUT
	nActionId	: UINT;
END_VAR
IF ActionDispacher.eCurrentState = E_MachineState.MACHINESTATE_Active THEN
	M_StopAction := ActionDispacher.M_StopAction(nActionId);
END_IF
END_METHOD

END_FUNCTION_BLOCK

// ---- OperatingModes/FB_OM_Auto.TcPOU
FUNCTION_BLOCK FB_OM_Auto
VAR_INPUT
END_VAR
VAR_OUTPUT
	eCurrentState 		: E_MachineState := E_MachineState.MACHINESTATE_Idle;
END_VAR
VAR
	pSequence		: POINTER TO FB_Sequence;	

	bError			: BOOL;
	stError			: ST_Error;
	i				: UINT;
	eLastState		: E_MachineState := E_MachineState.MACHINESTATE_Idle;
	
	nActionId		: UINT;
	
	nStateA_Reset : USINT;
	timeout : TON;
	
	nActActionsInPause : UDINT;
	
END_VAR

//Wenn der ActionDispacher in Error geht, dann alles abbrechen und in Error gehen
IF eCurrentState <> E_MachineState.MACHINESTATE_Reset THEN
	IF ActionDispacher.eCurrentState = E_MachineState.MACHINESTATE_Error THEN
		eCurrentState := E_MachineState.MACHINESTATE_Error;
		RETURN;
	END_IF
END_IF

CASE eCurrentState OF
	E_MachineState.MACHINESTATE_Idle:
		A_FillPCV();
		MEMSET(ADR(stInteractRequest),0,SIZEOF(stInteractRequest));
		MEMSET(ADR(stInterResponse),0,SIZEOF(stInterResponse));
		//Auf Fehler der Hardware reagieren und eventuelle CustomUnitType2 reagieren
		IF PerformHardware.bError OR fbObjectDirectory.M_CustomUnitType2_Error() THEN
			eCurrentState := E_MachineState.MACHINESTATE_Error;
		END_IF
		
	E_MachineState.MACHINESTATE_Running:
		//In diesem State wird solange gewartet, wie die SequenceAction fertig ist
		A_FillPCV();
		eLastState := E_MachineState.MACHINESTATE_Running;
		IF pSequence^.eCurrentState = E_SequenceState.State_Ready THEN
			eCurrentState := E_MachineState.MACHINESTATE_Ready;
		ELSIF pSequence^.eCurrentState = E_SequenceState.State_Canceled THEN
			eCurrentState := E_MachineState.MACHINESTATE_Ready;
		ELSIF pSequence^.eCurrentState = E_SequenceState.State_Pause THEN
			eCurrentState := E_MachineState.MACHINESTATE_Pause;
		ELSIF pSequence^.eCurrentState = E_SequenceState.State_Error THEN
			eCurrentState := E_MachineState.MACHINESTATE_Error;
		END_IF
		
		IF fbObjectDirectory.M_CustomUnitType2_Error() THEN
			ActionDispacher.M_StopAll();
			eCurrentState := E_MachineState.MACHINESTATE_Error;
		END_IF
		
		
	E_MachineState.MACHINESTATE_PauseRequest:
		IF pSequence^.eCurrentState = E_SequenceState.State_Pause THEN
			eCurrentState := E_MachineState.MACHINESTATE_Pause;
		ELSIF pSequence^.eCurrentState = E_SequenceState.State_Canceled THEN
			eCurrentState := E_MachineState.MACHINESTATE_Idle;
		END_IF
		
	E_MachineState.MACHINESTATE_Pause:
		A_FillPCV();
		//Aus diesem State kann in den ManualOverride gewechsel werden
		IF pSequence^.eCurrentState = E_SequenceState.State_Active THEN
			eCurrentState := E_MachineState.MACHINESTATE_Running;
		ELSIF pSequence^.eCurrentState = E_SequenceState.State_Canceled THEN
			eCurrentState := E_MachineState.MACHINESTATE_Idle;	
		ELSIF pSequence^.eCurrentState = E_SequenceState.State_Error THEN
			eCurrentState := E_MachineState.MACHINESTATE_Error;
		END_IF
	
	E_MachineState.MACHINESTATE_Active:
		A_FillPCV();
		IF eLastState = E_MachineState.MACHINESTATE_Idle THEN
			eCurrentState := ActionDispacher.eCurrentState;
		ELSIF eLastState = E_MachineState.MACHINESTATE_Pause THEN
			IF ActionDispacher.eCurrentState = E_MachineState.MACHINESTATE_Error THEN
				eCurrentState := E_MachineState.MACHINESTATE_Error;
			ELSE
				IF ActionDispacher.P_nActiveActions <= nActActionsInPause THEN //RunSequence bleibt aktiv
					eCurrentState := E_MachineState.MACHINESTATE_Pause;
				END_IF
			END_IF
		END_IF
		
		IF fbObjectDirectory.M_CustomUnitType2_Error() THEN
			ActionDispacher.M_StopAll();
			eCurrentState := E_MachineState.MACHINESTATE_Error;
		END_IF
		
		//In diesem Mode werden manuelle Actions ausgeführt
		//es sollte immer nur eine möglich sein
		//Hier besteht das Problem, dass einen in Pause gestellte Action, den ActionDispacher aktiv hält?
		//Testen!! Ja, so ist es
		//Am besten, man macht das über die ActionId und fragt diese ab, ob sie fertig ist
		
		(*IF fbActionDispacher.M_GetActionStatus(nActionId) = E_ActionStatus.ACTIONSTATUS_Ready THEN //Action fertig
			eCurrentState := E_MachineState.MACHINESTATE_Ready;
		END_IF*)
	
	E_MachineState.MACHINESTATE_Cancel:
				
	eCurrentState := ActionDispacher.eCurrentState;
	
	E_MachineState.MACHINESTATE_Canceled:
		eCurrentState := ActionDispacher.eCurrentState;
		
	E_MachineState.MACHINESTATE_Ready:
		//In diesem State wird der Head freigefahren
		IF eLastState = E_MachineState.MACHINESTATE_Running THEN
			eCurrentState := E_MachineState.MACHINESTATE_Idle;
			FOR i:= 1 TO UINT_TO_USINT(fbObjectDirectory.nCntMZHead) BY 1 DO
				IF afbMzHead[i].M_GetActionBusy(E_Action.ACTION_MoveZ) THEN
					eCurrentState := E_MachineState.MACHINESTATE_Ready;
				END_IF
			END_FOR
		ELSIF eLastState = E_MachineState.MACHINESTATE_Pause THEN
			eCurrentState := E_MachineState.MACHINESTATE_Pause;
		ELSIF eLastState = E_MachineState.MACHINESTATE_Idle THEN
			eCurrentState := E_MachineState.MACHINESTATE_Idle;	
		END_IF

	E_MachineState.MACHINESTATE_Reset:
		A_Reset();
	E_MachineState.MACHINESTATE_Error:
		//Do nothing
END_CASE

ACTION A_FillPCV:
IF (fbObjectDirectory.nCntPiezoPip > 0) OR (fbObjectDirectory.nCntSolenoidPip > 0) THEN
	fbPCV.M_Fill();
	IF fbPCV.bError THEN
		stError.HardwareGrp := E_HardwareGrp.PCV;
		stError.HardwareNr := 1;
		stError.MachineMode := E_MachineMode.MACHINEMODE_Manu;
		stError.POU := 1;
		stError.POUAction := E_POUACT.POUACT_UNDEFIEND;
		stError.ErrorId := fbPCV.nErrorId;
		fbErrorList.A_Add(putValue := stError);
		ActionDispacher.M_StopAll();
		eCurrentState := E_MachineState.MACHINESTATE_Error;
		RETURN;
	END_IF
END_IF
END_ACTION

ACTION A_Reset:
IF nStateA_Reset = 0 THEN
	timeout(IN:= FALSE);
	//ActionDispacher zurücksetzen (Hier werden auch die Devices zurückgesetzt
	ActionDispacher.M_Reset();
	//Hardware zurücksetzen
	PerformHardware.A_ResetError();
	//PCV zurücksetzen
	fbPCV.M_Reset();
	
	IF pSequence > 0 THEN
		pSequence^.M_Reset();	
	END_IF
		
	nStateA_Reset := 1;
ELSIF nStateA_Reset = 1 THEN
	nStateA_Reset := 2;
	timeout(IN:= TRUE, PT:=T#20S);
	//Warten, bis alles zurückgesetzt
	IF ActionDispacher.eCurrentState <> E_MachineState.MACHINESTATE_Idle THEN
		nStateA_Reset := 1; 		
	END_IF
	IF PerformHardware.bError THEN
		PerformHardware.A_ResetError();
		nStateA_Reset := 1;
	END_IF
	IF timeout.Q THEN
		eCurrentState := E_MachineState.MACHINESTATE_Error;
		nStateA_Reset := 0;
	END_IF
ELSIF nStateA_Reset = 2 THEN
	//Reset CustomUnitType2 (kann möglicherweise noch in Error stehen, weil evtl. ActionDispacher nicht in Error war)
	//Dadurch werden Objekte diesen Typs nicht durch den AD zurückgesetzt.
	fbObjectDirectory.M_ResetCustomUnitType2();
	
	//Checken, ob MzBase komplett resettet wurde -> Aktivierung der KOnfiguration erforderlich
	FOR i:= 1 TO fbObjectDirectory.nCntMZHead BY 1 DO
		IF aFbMultiZRef[i].P_bMzBaseRestarted THEN
			fbConfiguration.M_Deactivate();
		END_IF
	END_FOR
	
	IF fbConfiguration.P_bActivated THEN
		bError := FALSE;
		eLastState := E_MachineState.MACHINESTATE_Idle;
		eCurrentState := E_MachineState.MACHINESTATE_Idle;
		nStateA_Reset := 0;
	ELSE
		nStateA_Reset := 3;
	END_IF
ELSIF nStateA_Reset = 3 THEN //Konfiguration wieder aktivieren
	fbConfiguration.A_Activate(bExecute:= TRUE);
	IF NOT fbConfiguration.bBusy THEN
		IF fbConfiguration.bError THEN
			eCurrentState := E_MachineState.MACHINESTATE_Error;
			fbErrorList.M_Add(stError);
		ELSE
			bError := FALSE;
			eLastState := E_MachineState.MACHINESTATE_Idle;
			eCurrentState := E_MachineState.MACHINESTATE_Idle;
		END_IF
		nStateA_Reset := 0;
		fbConfiguration.A_Activate(bExecute:= FALSE);
	END_IF
END_IF
END_ACTION

METHOD M_Cancel : ERRORID
VAR_INPUT
END_VAR
IF 	eCurrentState =  E_MachineState.MACHINESTATE_Running OR
	eCurrentState =  E_MachineState.MACHINESTATE_PauseRequest OR
	eCurrentState =  E_MachineState.MACHINESTATE_Active OR
	eCurrentState =  E_MachineState.MACHINESTATE_Pause THEN
	ActionDispacher.M_StopAll();
	eCurrentState := E_MachineState.MACHINESTATE_Cancel;
END_IF
END_METHOD

METHOD M_ContinueAction : ERRORID
VAR_INPUT
	nActionId	: UINT;
END_VAR
IF eCurrentState = E_MachineState.MACHINESTATE_Pause THEN
	M_ContinueAction := ActionDispacher.M_ContinueAction(nActionId);
END_IF
END_METHOD

METHOD M_ExeAction : ERRORID
VAR_INPUT
	refActionData	: REFERENCE TO ST_ActionData;
END_VAR

VAR_OUTPUT
	nActionId		: UINT;
END_VAR

VAR
	nErrorId		: ERRORID;
END_VAR
CASE eCurrentState OF
	E_MachineState.MACHINESTATE_Idle:
		//folgende Actions können aus diesem heraus ausgeführt werden
		//-Programm löschen
		//-Programmschritt hochladen
		//-Condition hochladen
		//-Programm starten
		//-diverse Action ausführen (z.b. Druck,Temperatur ändern usw)
		//-Sequence starten
		nErrorId := ActionDispacher.M_ExeAction(refActionData:= refActionData,bExtern:= TRUE, nActionId=> nActionId);
		IF nErrorId > 0 THEN
			M_ExeAction := nErrorId;
			RETURN;
		ELSE
			eLastState := E_MachineState.MACHINESTATE_Idle;
			IF refActionData.eAction = E_Action.ACTION_RunSequence THEN
				pSequence := fbSequenceList.M_Get(DINT_TO_UDINT(refActionData.aParams[1]));
				eCurrentState := E_MachineState.MACHINESTATE_Running;
			ELSE
				eCurrentState := E_MachineState.MACHINESTATE_Active;
				ActionDispacher.P_bPauseRequestIntern := FALSE;
				ActionDispacher.P_bLastActionResult := FALSE;
			END_IF
		END_IF
		
	E_MachineState.MACHINESTATE_Active:
		//In disem State lässt sich keine Sequence starten
		IF refActionData.eAction = E_Action.ACTION_RunSequence THEN
			M_ExeAction := E_ErrorIdCmd.ERRORID_InvalidState;
			RETURN;
		END_IF
		nErrorId := ActionDispacher.M_ExeAction(refActionData:= refActionData,bExtern:= TRUE, nActionId=> nActionId);
		//-diverse Action ausführen (z.b. Druck,Temperatur ändern usw)
	E_MachineState.MACHINESTATE_Pause:
		//In Pause können im Grunde alle Actions außer RunGCode usw. ausgeführt werden
		//allerdings darf, während eine Action aktiv ist, kein Continue erfolgen
		(*CASE refActionData.eAction OF
			
		END_CASE
			E_Action.ACTION_Cooling, E_Action.ACTION_Heating, E_Action.ACTION_InkOpClCover, E_Action.ACTION_InkSpin,
			E_Action.ACTION_MoveZ, E_Action.ACTION_ReactorOpCl, E_Action.ACTION_SetPressure, E_Action.ACTION_SetVoltage,
			E_Action.ACTION_SwitchLight, E_Action.ACTION_SwitchPressure, E_Action.ACTION_SwitchVoltage, E_Action.ACTION_CleanTip:
			
			nErrorId := fbActionDispacher.M_ExeAction(refActionData:= refActionData,bInfo:= TRUE, nActionId=> nActionId);
		ELSE
			M_ExeAction := E_ErrorIdCmd.ERRORID_InvalidState;
			RETURN;
		END_CASE*)
		IF refActionData.eAction > 50 THEN
			
			M_ExeAction := ActionDispacher.M_ExeAction(refActionData:= refActionData,bExtern:= TRUE, nActionId=> nActionId);
			IF 	M_ExeAction = 0 THEN
				eLastState := E_MachineState.MACHINESTATE_Pause;
				eCurrentState := E_MachineState.MACHINESTATE_Active;
				nActActionsInPause := ActionDispacher.P_nActiveActions - 1;	
			END_IF
		ELSE
			M_ExeAction := E_ErrorIdCmd.ERRORID_InvalidState;
			RETURN;
		END_IF

	E_MachineState.MACHINESTATE_Running:
		IF refActionData.eAction = E_Action.ACTION_SetPressure OR refActionData.eAction = E_Action.ACTION_DispenseDrops THEN
			nErrorId := ActionDispacher.M_ExeAction(refActionData:= refActionData,bExtern:= TRUE, nActionId=> nActionId);
		ELSE
			M_ExeAction := E_ErrorIdCmd.ERRORID_InvalidState;
			RETURN;
		END_IF
ELSE
	//Actions verschiedene Fehlermeldung zurückgeben!!!!
	M_ExeAction := E_ErrorIdCmd.ERRORID_InvalidState;
	RETURN;	
END_CASE
END_METHOD

METHOD M_PauseAction : ERRORID
VAR_INPUT
	nActionId	: UINT;
END_VAR
IF eCurrentState = E_MachineState.MACHINESTATE_Running THEN
	eLastState := E_MachineState.MACHINESTATE_Running;
	ActionDispacher.M_PauseAction(nActionId);
	eCurrentState := E_MachineState.MACHINESTATE_PauseRequest;
ELSIF eCurrentState = E_MachineState.MACHINESTATE_Active THEN
	eLastState := E_MachineState.MACHINESTATE_Active;
	ActionDispacher.M_PauseAction(nActionId);
ELSE
	M_PauseAction := E_ErrorIdCmd.ERRORID_InvalidState;
END_IF
END_METHOD

METHOD M_ResetError
VAR_INPUT
END_VAR
IF eCurrentState = E_MachineState.MACHINESTATE_Error THEN
	eCurrentState := E_MachineState.MACHINESTATE_Reset;
END_IF
END_METHOD

METHOD M_StopAction : ERRORID
VAR_INPUT
	nActionId	: UINT;
END_VAR
M_StopAction := ActionDispacher.M_StopAction(nActionId);
END_METHOD

END_FUNCTION_BLOCK

// ---- OperatingModes/FB_OM_SemiAuto.TcPOU
FUNCTION_BLOCK FB_OM_SemiAuto
VAR_INPUT
END_VAR
VAR_OUTPUT
	eCurrentState : E_MachineState := E_MachineState.MACHINESTATE_Idle;
END_VAR
VAR
	nCalls	: UINT;
END_VAR

nCalls := nCalls + 1;

METHOD M_ResetError
VAR_INPUT
END_VAR
END_METHOD

END_FUNCTION_BLOCK

// ---- OperatingModes/FB_OM_Maintenance.TcPOU
FUNCTION_BLOCK FB_OM_Maintenance
VAR_INPUT
END_VAR
VAR_OUTPUT
	eCurrentState : E_MachineState := E_MachineState.MACHINESTATE_Idle;
END_VAR
VAR
	bError					: BOOL;
	stError					: ST_Error;
	nErrorId				: ERRORID;
	bDeviceFirmwUpdate		: BOOL;
	nStateAction			: UINT;
	pFbCanNode				: POINTER TO FB_CanNodeBase;

	bSetupXYAxis			: BOOL;
	pSetupDrive				: POINTER TO FB_XYDriveBase;
	bSetupZAxis				: BOOL;
	pFbZAxis				: POINTER TO FB_ZAxisRef;
	pFbMultiZ				: POINTER TO FB_MultiZRef;
	fbZmHome				: FB_ZM_Home;
	
	nStateA_Reset 			: USINT;
	
	//ResetPlc
	bResetPlc				: BOOL;
	nStateA_ResetPlc 		: USINT;
	fbPLC_Reset				: PLC_Reset;
	
	timeout : TON;
	
	i : USINT;
	
END_VAR

IF bResetPlc THEN
	A_ResetPlc();
	RETURN;	//andere Actions werden nicht mehr ausgeführt!
END_IF

IF eCurrentState = E_MachineState.MACHINESTATE_Active THEN
	
	IF bDeviceFirmwUpdate THEN	//FirmwareUpdate Can-Nodes
		A_DeviceFirmwUpdate();
	ELSIF bSetupXYAxis THEN	//Achsen einrichten (Referenzpunkt usw. bestimmen)
		A_SetupXYAxis();
	ELSIF bSetupZAxis THEN	//Achsen einrichten (Referenzpunkt usw. bestimmen)
		A_SetupZAxis();
	ELSE
		eCurrentState := ActionDispacher.eCurrentState;	
	END_IF
	
	IF nStateAction >= 80 THEN
		IF nStateAction >= 99 THEN
			bError := TRUE;
			fbErrorList.M_Add(stError);
		END_IF
		bDeviceFirmwUpdate := FALSE;
		bSetupXYAxis := FALSE;
		bSetupZAxis := FALSE;
		nStateAction := 0;
	END_IF

	IF bError THEN
		eCurrentState := E_MachineState.MACHINESTATE_Error;
		RETURN;
	END_IF
	
	IF NOT (bDeviceFirmwUpdate OR bSetupXYAxis OR bSetupZAxis) THEN
		eCurrentState := E_MachineState.MACHINESTATE_Idle;
	END_IF
	
ELSIF eCurrentState = E_MachineState.MACHINESTATE_Reset THEN
	A_Reset();
END_IF

ACTION A_DeviceFirmwUpdate:
CASE nStateAction OF
	0:
		FirmwUpdate.pFbCanNode := pFbCanNode;
		FirmwUpdate.bExecute := TRUE;
		nStateAction := 1;
	
	1:
		IF NOT FirmwUpdate.bBusy THEN
			IF FirmwUpdate.bError THEN
				stError.ErrorId := FirmwUpdate.nErrorId;
				nStateAction := 99;
			ELSE
				nStateAction := 80;
			END_IF
			FirmwUpdate.bExecute := FALSE;
		END_IF
END_CASE
END_ACTION

ACTION A_Reset:
IF nStateA_Reset = 0 THEN
	//ActionDispacher zurücksetzen (Hier werden auch die Devices zurückgesetzt
	ActionDispacher.M_Reset();
	//Hardware zurücksetzen
	PerformHardware.A_ResetError();
	//PCV zurücksetzen
	fbPCV.M_Reset();
	timeout(IN:= FALSE);
	nStateA_Reset := 1;
ELSIF nStateA_Reset = 1 THEN
	nStateA_Reset := 2;
	timeout(IN:= TRUE, PT:=T#20S);
	//Warten, bis alles zurückgesetzt
	IF ActionDispacher.eCurrentState <> E_MachineState.MACHINESTATE_Idle THEN
		nStateA_Reset := 1; 		
	END_IF
	IF PerformHardware.bError THEN
		PerformHardware.A_ResetError();
		nStateA_Reset := 1;
	END_IF
	IF timeout.Q THEN
		eCurrentState := E_MachineState.MACHINESTATE_Error;
		nStateA_Reset := 0;
	END_IF
ELSIF nStateA_Reset = 2 THEN
	bError := FALSE;
	eCurrentState := E_MachineState.MACHINESTATE_Idle;
	nStateA_Reset := 0;
END_IF
END_ACTION

ACTION A_ResetPlc:
CASE nStateA_ResetPlc OF
	0:	//Alle MzHeads resetten
		FOR i:= 1 TO cMaxMzHeads BY 1 DO
			aFbMultiZRef[i].M_ResetApp();
		END_FOR
		nStateA_ResetPlc := 1;
		
	1:	//warten, bis mind 1 NodeState <> 0
		FOR i:= 1 TO cMaxMzHeads BY 1 DO
			IF aFbMultiZRef[i].P_nNodeState <> 0 THEN
				nStateA_ResetPlc := 2;	
			END_IF
		END_FOR
	
	2:	//warten bis sich alle MzHeads wieder melden (Timeout)
		timeout(IN:=TRUE, PT:=T#6S);
		nStateA_ResetPlc := 3;
		FOR i:= 1 TO cMaxMzHeads BY 1 DO
			IF aFbMultiZRef[i].P_nNodeState <> 0 THEN
				nStateA_ResetPlc := 2;	
			END_IF
		END_FOR
		IF timeout.Q THEN
			nStateA_ResetPlc := 3;
		END_IF
	
	3:	//Plc resetten
		fbPLC_Reset(PORT:= 851, RESET:= TRUE);
END_CASE
END_ACTION

ACTION A_SetupXYAxis:
CASE nStateAction OF
	0:	
		stError.ErrorId :=  pSetupDrive^.M_Setup();
		IF stError.ErrorId > 0 THEN
			nStateAction := 99;
		ELSE
			MEMSET(ADR(stInterResponse),0,SIZEOF(stInterResponse));
			nStateAction := 1;
		END_IF
	
	1:	//Warten, bis Axis auf UserResponse wartet	
		IF pSetupDrive^.P_bError THEN
			stError.ErrorId := pSetupDrive^.P_nErrorId;
			nStateAction := 99;
		ELSE
			IF pSetupDrive^.P_bSetupWaitForResp THEN
				MEMSET(ADR(stInterResponse),0,SIZEOF(stInterResponse));
				stInteractRequest.eInteractMessageType := E_InteractMessageType.INTERACTMES_StartTeaching;	//Interaction Request absenden
				nStateAction := 2;
			ELSE
				//auf Cancel reagieren
				IF stInterResponse.eInteractMessageType = E_InteractMessageType.INTERACTMES_Cancel THEN
					nStateAction := 70;	
				END_IF
			END_IF
		END_IF
		
	2:	//auf Response von PC warten
		IF stInterResponse.eInteractMessageType = E_InteractMessageType.INTERACTMES_TeachingFinished THEN
			MEMSET(ADR(stInteractRequest),0,SIZEOF(stInteractRequest));
			pSetupDrive^.M_ContinueSetup();
			nStateAction := 3;
		ELSIF stInterResponse.eInteractMessageType = E_InteractMessageType.INTERACTMES_Cancel THEN
			nStateAction := 70;
		END_IF
	3:
		IF NOT pSetupDrive^.P_bBusy THEN
			fbSettings.M_WritePersData();
			nStateAction := 80;
		END_IF
		
	70:	//Abbrechen
		pSetupDrive^.M_Stop();
		MEMSET(ADR(stInteractRequest),0,SIZEOF(stInteractRequest));
		nStateAction := 80;
		
END_CASE
END_ACTION

ACTION A_SetupZAxis:
IF nStateAction = 0 THEN
	fbZmHome(bExecute:= TRUE, pFbZAxisRef:= pFbZAxis, bMoveToHome:= FALSE);
	IF NOT fbZmHome.bBusy THEN
		IF fbZmHome.bError THEN
			nStateAction := 99;
		ELSE
			MEMSET(ADR(stInterResponse),0,SIZEOF(stInterResponse));
			stInteractRequest.eInteractMessageType := E_InteractMessageType.INTERACTMES_StartTeaching;	
			nStateAction := 1;
		END_IF
		fbZmHome(bExecute:= FALSE);
	END_IF
ELSIF nStateAction = 1 THEN //auf Response von PC warten
	IF stInterResponse.eInteractMessageType = E_InteractMessageType.INTERACTMES_TeachingFinished THEN
		MEMSET(ADR(stInteractRequest),0,SIZEOF(stInteractRequest));
		pFbZAxis^.P_rRefPos := DINT_TO_REAL(stInterResponse.nArg1);
		fbSettings.M_WritePersData();
		nStateAction := 80;
	ELSIF stInterResponse.eInteractMessageType = E_InteractMessageType.INTERACTMES_Cancel THEN
		MEMSET(ADR(stInteractRequest),0,SIZEOF(stInteractRequest));
		nStateAction := 80;
	END_IF
ELSIF nStateAction = 70 THEN
	nStateAction := 80;	
END_IF
END_ACTION

METHOD M_Cancel : ERRORID
VAR_INPUT
END_VAR
VAR
END_VAR
IF eCurrentState = E_MachineState.MACHINESTATE_Active THEN	//auf Cancel-Kommando braucht nur im Actice-State reagiert werden
	IF bSetupXYAxis OR bSetupZAxis THEN
		nStateAction := 70;
	END_IF
END_IF
END_METHOD

METHOD M_DeviceFirmwUpdate : ERRORID
VAR_INPUT
	nCanNodeId	: USINT;
END_VAR
IF eCurrentState = E_MachineState.MACHINESTATE_Idle OR eCurrentState = E_MachineState.MACHINESTATE_Error THEN
	//Folgende CAN-Knoten (Gesim) können upgedatet werden
	//MultiZ, ReactorHeater, MtpHeater, SubstHeater, BottleRack, IOPortExpander
	pFbCanNode := 0;
	CASE nCanNodeId OF
		5:	//ReactorHeater1
			{IF defined(variable:aFbReactHeatRef)}
			pFbCanNode := ADR(aFbReactHeatRef[1]);
			{END_IF}
		6:	//ReactorHeater2
			{IF defined(variable:aFbReactHeatRef)}
			IF cNoOfReactHeaters > 1 THEN
				pFbCanNode := ADR(aFbReactHeatRef[1]) + SIZEOF(aFbReactHeatRef[1]);
			END_IF
			{END_IF}
		8:	//MultiZ1
			{IF defined(variable:aFbMultiZRef)}
			pFbCanNode := ADR(aFbMultiZRef[1]);
			{END_IF}
		9:	//MultiZ2
			{IF defined(variable:aFbMultiZRef)}
			IF cMaxMzHeads > 1 THEN
				pFbCanNode := ADR(aFbMultiZRef[1]) + SIZEOF(aFbMultiZRef[1]);	
			END_IF
			{END_IF}
		10:	//MtpHeater1
			{IF defined(variable:aFbMtpHeatRef)}
			pFbCanNode := ADR(aFbMtpHeatRef[1]);
			{END_IF}
		11:	//MtpHeater2
			{IF defined(variable:aFbMtpHeatRef)}
			IF cNoOfMtpHeaters > 1 THEN
				pFbCanNode := ADR(aFbMtpHeatRef[1]) + SIZEOF(aFbMtpHeatRef[1]);
			END_IF
			{END_IF}
		12:	//SubstHeater1
			{IF defined(variable:aFbSubstHeatRef)}
			pFbCanNode := ADR(aFbSubstHeatRef[1]);
			{END_IF}
		13:	//SubstHeater2
			{IF defined(variable:aFbSubstHeatRef)}
			IF cNoOfSubstHeaters > 1 THEN
				pFbCanNode := ADR(aFbSubstHeatRef[1]) + SIZEOF(aFbSubstHeatRef[1]);
			END_IF
			{END_IF}
		14:	//TripleTrigger1
			{IF defined(variable:aFbTripleTriggerRef)}
			pFbCanNode := ADR(aFbTripleTriggerRef[1]);
			{END_IF}		
		16:	//IOExpander1
			{IF defined(variable:aFbIOExpanderRef)}
			pFbCanNode := ADR(aFbIOExpanderRef[1]);
			{END_IF}		
		17:	//IOExpander2
			{IF defined(variable:aFbIOExpanderRef)}
			IF cNoOfIOExpanders > 1 THEN
				pFbCanNode := ADR(aFbIOExpanderRef[1]) + SIZEOF(aFbIOExpanderRef[1]);
			END_IF
			{END_IF}		
		20:	//BottleRack1
			{IF defined(variable:aFbBottleRackRef)}
			pFbCanNode := ADR(aFbBottleRackRef[1]);
			{END_IF}			
		24:	//PowderStation1
			{IF defined(variable:aFbPowderStatRef)}
			pFbCanNode := ADR(aFbPowderStatRef[1]);
			{END_IF}
		25:	//MultiPurpIO
			{IF defined(variable:aFbHwRefMultiPurpIO)}
			pFbCanNode := ADR(aFbHwRefMultiPurpIO[1]);
			{END_IF}		
	END_CASE

	bDeviceFirmwUpdate := TRUE;
	eCurrentState := E_MachineState.MACHINESTATE_Active;
ELSE
	M_DeviceFirmwUpdate := E_ErrorIdCmd.ERRORID_InvalidState; 
END_IF
END_METHOD

METHOD M_ResetError
VAR_INPUT
END_VAR
IF eCurrentState = E_MachineState.MACHINESTATE_Error THEN 
	eCurrentState := E_MachineState.MACHINESTATE_Reset;
END_IF
END_METHOD

METHOD M_ResetPlc : ERRORID
VAR_INPUT
END_VAR
bResetPlc := TRUE;
END_METHOD

METHOD M_SetState
VAR_INPUT
	eState : E_MachineState;
END_VAR
eCurrentState := eState;
END_METHOD

METHOD M_SetupAxis : ERRORID
VAR_INPUT
	refCmdData : REFERENCE TO ST_CmdData;
END_VAR

VAR
	stHardwareId : ST_HardwareId;
END_VAR
IF eCurrentState <> E_MachineState.MACHINESTATE_Idle THEN
	M_SetupAxis := E_ErrorIdCmd.ERRORID_InvalidState;
	RETURN;
END_IF

IF NOT (pFbSafety^.eCurrentState = E_SafetyState.Locked) THEN
	M_SetupAxis := E_ErrorIdCmd.ERRORID_InterlockNotLocked;
	RETURN;	
END_IF

MEMCPY(ADR(stHardwareId),ADR(refCmdData.n32Data[0]),3);

IF stHardwareId.eGroup = E_HardwareGrp.AxisX OR stHardwareId.eGroup = E_HardwareGrp.AxisY THEN
	pSetupDrive := fbXYDriveList.M_GetByHwId(stHardwareId);
	IF pSetupDrive > 0 THEN
		pSetupDrive^.M_SetProperties(refCmdData);
		bSetupXYAxis := TRUE;	
	ELSE
		M_SetupAxis := E_ErrorIdCmd.ERRORID_InvalidHwItem;
	END_IF

ELSIF stHardwareId.eGroup = E_HardwareGrp.AxisZ THEN
	IF stHardwareId.nItem > 0 AND stHardwareId.nItem <= 7 THEN
		//Parent?
		IF stHardwareId.nParentItem > 0 AND stHardwareId.nParentItem <= cMaxMzHeads THEN
			pFbMultiZ := ADR(aFbMultiZRef[stHardwareId.nParentItem]);
			IF pFbMultiZ^.aFbZAxisRef[stHardwareId.nItem].stInput.nStatus.7 THEN
				pFbZAxis := ADR(pFbMultiZ^.aFbZAxisRef[stHardwareId.nItem]);
				pFbZAxis^.P_bInvertInitDir := DINT_TO_BOOL(refCmdData.n32Data[5]);
				bSetupZAxis := TRUE;
			ELSE
				M_SetupAxis := E_ErrorIdMultiZ.ERRORID_NoZAxis;	
			END_IF
		ELSE
			M_SetupAxis := E_ErrorIdCmd.ERRORID_InvalidHwItem;
		END_IF
	ELSE
		M_SetupAxis := E_ErrorIdCmd.ERRORID_InvalidHwItem;
	END_IF
ELSE
	M_SetupAxis := E_ErrorIdCmd.ERRORID_InvalidHwGroup;
END_IF

IF M_SetupAxis = 0 THEN
	eCurrentState := E_MachineState.MACHINESTATE_Active;	
END_IF
END_METHOD

END_FUNCTION_BLOCK

// ---- Objects/Targets/Passive/FB_DryPad.TcPOU
FUNCTION_BLOCK FB_DryPad EXTENDS FB_TargetBase
VAR_INPUT
END_VAR

VAR_OUTPUT
	nCol 	: USINT;
	nRow 	: USINT;
END_VAR

VAR
	nNotifyId 				: UINT;
	stArea1Point1 			: ST_2DPoint;
	stArea1Point2 			: ST_2DPoint;
 	nArea1IntermedPointsX 	: UINT;
	nArea1IntermedPointsY 	: UINT;
	nArea1CountPoints		: UINT;
	stArea2Point1 			: ST_2DPoint;
	stArea2Point2 			: ST_2DPoint;
 	nArea2IntermedPointsX 	: UINT;
	nArea2IntermedPointsY 	: UINT;
	nArea2CountPoints		: UINT;
	nGCodeTargetNr			: UINT;
END_VAR

VAR PERSISTENT
	nCurrentColArea1		: USINT;
	nCurrentRowArea1		: USINT;
	nCurrentColArea2		: USINT;
	nCurrentRowArea2		: USINT;
END_VAR

METHOD FB_init : BOOL
VAR_INPUT
	bInitRetains : BOOL; // if TRUE, the retain variables are initialized (warm start / cold start)
	bInCopyCode : BOOL;  // if TRUE, the instance afterwards gets moved into the copy code (online change)
END_VAR
eObjectType := E_ObjectType.OBJECTTYPE_DryPad;
eObjectGroup := E_ObjectGroup.OBJECTGROUP_Target;
END_METHOD

METHOD M_AddChild : ERRORID
VAR_INPUT
	pObject	: POINTER TO FB_Object;
	nSlotNr	: UINT;
	nIndex 	: INT;
END_VAR
//Kann folgende Objekte aufnehmen:
//Point
IF pObject > 0 THEN
	IF pObject^.P_eObjectType = E_ObjectType.OBJECTTYPE_Point THEN
		M_AddChild := SUPER^.M_AddChild(pObject,nSlotNr,nIndex);
	ELSE
		M_AddChild := E_ErrorIdObjMgmt.ERRORID_InvalidParentObject;
	END_IF
ELSE
	M_AddChild := E_ErrorIdObjMgmt.ERRORID_InvalidParentObject;
END_IF
END_METHOD

METHOD M_CalcNextPosData
VAR_INPUT
	nArea : USINT;
END_VAR
IF nArea = 1 THEN
	//nächste Spalte ermitteln
	IF (nCurrentColArea1 = 0) OR (nCurrentColArea1 >= nArea1IntermedPointsX + 2) THEN
		nCurrentColArea1 := 1;
	ELSE
		nCurrentColArea1 := nCurrentColArea1 + 1;
	END_IF
	
	IF nCurrentColArea1 = 1 THEN
		//nächste Zeile ermitteln
		IF (nCurrentRowArea1 = 0) OR (nCurrentRowArea1 >= nArea1IntermedPointsY + 2) THEN
			nCurrentRowArea1 := 1;
		ELSE
			nCurrentRowArea1 := nCurrentRowArea1 + 1;
		END_IF
	END_IF
	
	nCol := nCurrentColArea1;
	nRow := nCurrentRowArea1;
	M_UpdateProcessData();
	//fbSettings.bWritePersitentData := TRUE;

ELSIF nArea = 2 THEN
	//nächste Spalte ermitteln
	IF (nCurrentColArea2 = 0) OR (nCurrentColArea2 >= nArea2IntermedPointsX + 2) THEN
		nCurrentColArea2 := 1;
	ELSE
		nCurrentColArea2 := nCurrentColArea2 + 1;
	END_IF
	
	IF nCurrentColArea2 = 1 THEN
		//nächste Zeile ermitteln
		IF (nCurrentRowArea2 = 0) OR (nCurrentRowArea2 >= nArea2IntermedPointsY + 2) THEN
			nCurrentRowArea2 := 1;
		ELSE
			nCurrentRowArea2 := nCurrentRowArea2 + 1;
		END_IF
	END_IF
	
	nCol := nCurrentColArea2;
	nRow := nCurrentRowArea2;	
	M_UpdateProcessData();
	//fbSettings.bWritePersitentData := TRUE;
END_IF
END_METHOD

METHOD M_ChangeCleanMat
VAR_INPUT
END_VAR
nCurrentColArea1 := 0;
nCurrentRowArea1 := 0;
nCurrentColArea2 := 0;
nCurrentRowArea2 := 0;
M_UpdateProcessData();
END_METHOD

METHOD M_CheckProps : ERRORID
VAR_INPUT
END_VAR
M_CheckProps := SUPER^.M_CheckProps();

IF M_CheckProps = 0 THEN
	M_UpdateProcessData();
END_IF
END_METHOD

